LIN {X 0,Y 230.578,Z 317.111,A -85,B 0,C 180,E1 -20760.813,E2 -20760.813} C_VEL
LIN {X 0,Y 233.907,Z 325.789,A -85,B 0,C 180,E1 -20762.609,E2 -20762.609} C_VEL
LIN {X 0,Y 238.982,Z 335.486,A -85,B 0,C 180,E1 -20765.008,E2 -20765.008} C_VEL
LIN {X 0,Y 245.081,Z 344.302,A -85,B 0,C 180,E1 -20767.553,E2 -20767.553} C_VEL
LIN {X 0,Y 253.175,Z 353.284,A -85,B 0,C 180,E1 -20770.543,E2 -20770.543} C_VEL
LIN {X 0,Y 261.948,Z 361.164,A -85,B 0,C 180,E1 -20773.525,E2 -20773.525} C_VEL
LIN {X 0,Y 271.147,Z 368.091,A -85,B 0,C 180,E1 -20776.51,E2 -20776.51} C_VEL
LIN {X 0,Y 276.4,Z 371.69,A -85,B 0,C 180,E1 -20778.264,E2 -20778.264} C_VEL
LIN {X 0,Y 283.012,Z 376.04,A -85,B 0,C 180,E1 -20780.657,E2 -20780.657} C_VEL
LIN {X 0,Y 288.749,Z 379.536,A -85,B 0,C 180,E1 -20783.01,E2 -20783.01} C_VEL
LIN {X 0,Y 291.205,Z 381.266,A -85,B 0,C 180,E1 -20784.46,E2 -20784.46} C_VEL
LIN {X 0,Y 293.286,Z 382.591,A -85,B 0,C 180,E1 -20785.878,E2 -20785.878} C_VEL
LIN {X 0,Y 295.421,Z 383.606,A -85,B 0,C 180,E1 -20787.399,E2 -20787.399} C_VEL
LIN {X 0,Y 296.734,Z 384.085,A -85,B 0,C 180,E1 -20788.643,E2 -20788.643} C_VEL
LIN {X 0,Y 297.612,Z 384.263,A -85,B 0,C 180,E1 -20790,E2 -20790} C_VEL
LIN {X 0,Y 296.714,Z 384.086,A -85,B 0,C 180,E1 -20791.357,E2 -20791.357} C_VEL
LIN {X 0,Y 295.23,Z 383.531,A -85,B 0,C 180,E1 -20792.729,E2 -20792.729} C_VEL
LIN {X 0,Y 293.276,Z 382.591,A -85,B 0,C 180,E1 -20794.123,E2 -20794.123} C_VEL
LIN {X 0,Y 289.886,Z 380.295,A -85,B 0,C 180,E1 -20796.383,E2 -20796.383} C_VEL
LIN {X 0,Y 287.004,Z 378.499,A -85,B 0,C 180,E1 -20797.74,E2 -20797.74} C_VEL
LIN {X 0,Y 281.117,Z 374.761,A -85,B 0,C 180,E1 -20800.078,E2 -20800.078} C_VEL
LIN {X 0,Y 273.672,Z 369.778,A -85,B 0,C 180,E1 -20802.671,E2 -20802.671} C_VEL
LIN {X 0,Y 265.413,Z 363.851,A -85,B 0,C 180,E1 -20805.354,E2 -20805.354} C_VEL
LIN {X 0,Y 255.737,Z 355.726,A -85,B 0,C 180,E1 -20808.579,E2 -20808.579} C_VEL
LIN {X 0,Y 247.025,Z 346.636,A -85,B 0,C 180,E1 -20811.706,E2 -20811.706} C_VEL
LIN {X 0,Y 241.827,Z 339.902,A -85,B 0,C 180,E1 -20813.764,E2 -20813.764} C_VEL
LIN {X 0,Y 236.613,Z 331.326,A -85,B 0,C 180,E1 -20816.068,E2 -20816.068} C_VEL
LIN {X 0,Y 232.585,Z 322.649,A -85,B 0,C 180,E1 -20818.071,E2 -20818.071} C_VEL
LIN {X 0,Y 229.455,Z 313.908,A -85,B 0,C 180,E1 -20819.786,E2 -20819.786} C_VEL
LIN {X 0,Y 225.733,Z 303.804,A -85,B 0,C 180,E1 -20821.564,E2 -20821.564} C_VEL
LIN {X 0,Y 220.845,Z 293.133,A -85,B 0,C 180,E1 -20823.371,E2 -20823.371} C_VEL
LIN {X 0,Y 216.792,Z 285.655,A -85,B 0,C 180,E1 -20824.644,E2 -20824.644} C_VEL
LIN {X 0,Y 215.273,Z 282.957,A -85,B 0,C 180,E1 -20825.085,E2 -20825.085} C_VEL
LIN {X 0,Y 213.929,Z 280.441,A -85,B 0,C 180,E1 -20825.467,E2 -20825.467} C_VEL
LIN {X 0,Y 213.702,Z 279.367,A -85,B 0,C 180,E1 -20825.598,E2 -20825.598} C_VEL
LIN {X 0,Y 213.74,Z 279.361,A -85,B 0,C 180,E1 -20828.662,E2 -20828.662} C_VEL
LIN {X 0,Y 213.756,Z 279.358,A -85,B 0,C 180,E1 -20831.114,E2 -20831.114} C_VEL
LIN {X 0,Y 213.798,Z 279.354,A -85,B 0,C 180,E1 -20833.701,E2 -20833.701} C_VEL
LIN {X 0,Y 213.775,Z 279.356,A -85,B 0,C 180,E1 -20836.358,E2 -20836.358} C_VEL
LIN {X 0,Y 213.762,Z 279.358,A -85,B 0,C 180,E1 -20839.128,E2 -20839.128} C_VEL
LIN {X 0,Y 213.721,Z 279.363,A -85,B 0,C 180,E1 -20843.724,E2 -20843.724} C_VEL
LIN {X 0,Y 213.732,Z 279.361,A -85,B 0,C 180,E1 -20848.272,E2 -20848.272} C_VEL
LIN {X 0,Y 213.801,Z 279.352,A -85,B 0,C 180,E1 -20852.614,E2 -20852.614} C_VEL
LIN {X 0,Y 213.778,Z 279.355,A -85,B 0,C 180,E1 -20856.997,E2 -20856.997} C_VEL
LIN {X 0,Y 213.866,Z 279.345,A -85,B 0,C 180,E1 -20862.81,E2 -20862.81} C_VEL
LIN {X 0,Y 213.916,Z 279.336,A -85,B 0,C 180,E1 -20866.716,E2 -20866.716} C_VEL
LIN {X 0,Y 214.123,Z 279.307,A -85,B 0,C 180,E1 -20870.566,E2 -20870.566} C_VEL
LIN {X 0,Y 214.079,Z 279.318,A -85,B 0,C 180,E1 -20874.359,E2 -20874.359} C_VEL
LIN {X 0,Y 214.434,Z 279.246,A -85,B 0,C 180,E1 -20878.133,E2 -20878.133} C_VEL
LIN {X 0,Y 214.534,Z 279.246,A -85,B 0,C 180,E1 -20880.011,E2 -20880.011} C_VEL
LIN {X 0,Y 214.403,Z 279.274,A -85,B 0,C 180,E1 -20881.889,E2 -20881.889} C_VEL
LIN {X 0,Y 214.185,Z 279.305,A -85,B 0,C 180,E1 -20887.552,E2 -20887.552} C_VEL
LIN {X 0,Y 213.994,Z 279.33,A -85,B 0,C 180,E1 -20891.375,E2 -20891.375} C_VEL
LIN {X 0,Y 213.901,Z 279.342,A -85,B 0,C 180,E1 -20895.25,E2 -20895.25} C_VEL
LIN {X 0,Y 213.802,Z 279.353,A -85,B 0,C 180,E1 -20899.201,E2 -20899.201} C_VEL
LIN {X 0,Y 213.795,Z 279.355,A -85,B 0,C 180,E1 -20903.243,E2 -20903.243} C_VEL
LIN {X 0,Y 213.805,Z 279.532,A -85,B 0,C 180,E1 -20907.439,E2 -20907.439} C_VEL
LIN {X 0,Y 214.004,Z 281.177,A -85,B 0,C 180,E1 -20911.709,E2 -20911.709} C_VEL
LIN {X 0,Y 214.25,Z 283.111,A -85,B 0,C 180,E1 -20916.2,E2 -20916.2} C_VEL
LIN {X 0,Y 214.622,Z 285.39,A -85,B 0,C 180,E1 -20920.925,E2 -20920.925} C_VEL
LIN {X 0,Y 214.75,Z 286.989,A -85,B 0,C 180,E1 -20923.949,E2 -20923.949} C_VEL
LIN {X 0,Y 214.684,Z 288.477,A -85,B 0,C 180,E1 -20926.571,E2 -20926.571} C_VEL
LIN {X 0,Y 214.492,Z 289.965,A -85,B 0,C 180,E1 -20929.058,E2 -20929.058} C_VEL
LIN {X 0,Y 213.761,Z 292.894,A -85,B 0,C 180,E1 -20933.716,E2 -20933.716} C_VEL
LIN {X 0,Y 213.629,Z 293.565,A -85,B 0,C 180,E1 -20934.675,E2 -20934.675} C_VEL
LIN {X 0,Y 214.491,Z 296.709,A -85,B 0,C 180,E1 -20935.014,E2 -20935.014} C_VEL
LIN {X 0,Y 218.05,Z 307.158,A -85,B 0,C 180,E1 -20936.47,E2 -20936.47} C_VEL
LIN {X 0,Y 221.031,Z 319.519,A -85,B 0,C 180,E1 -20938.304,E2 -20938.304} C_VEL
LIN {X 0,Y 222.724,Z 329.353,A -85,B 0,C 180,E1 -20939.908,E2 -20939.908} C_VEL
LIN {X 0,Y 223.702,Z 338.852,A -85,B 0,C 180,E1 -20941.618,E2 -20941.618} C_VEL
LIN {X 0,Y 223.928,Z 348.013,A -85,B 0,C 180,E1 -20943.452,E2 -20943.452} C_VEL
LIN {X 0,Y 223.641,Z 352.493,A -85,B 0,C 180,E1 -20944.4,E2 -20944.4} C_VEL
LIN {X 0,Y 220.928,Z 362.07,A -85,B 0,C 180,E1 -20946.57,E2 -20946.57} C_VEL
LIN {X 0,Y 218.712,Z 369.736,A -85,B 0,C 180,E1 -20948.75,E2 -20948.75} C_VEL
LIN {X 0,Y 216.744,Z 376.438,A -85,B 0,C 180,E1 -20951.08,E2 -20951.08} C_VEL
LIN {X 0,Y 215.21,Z 381.639,A -85,B 0,C 180,E1 -20953.264,E2 -20953.264} C_VEL
LIN {X 0,Y 213.669,Z 384.495,A -85,B 0,C 180,E1 -20954.603,E2 -20954.603} C_VEL
LIN {X 0,Y 209.677,Z 388.477,A -85,B 0,C 180,E1 -20956.803,E2 -20956.803} C_VEL
LIN {X 0,Y 205.968,Z 391.837,A -85,B 0,C 180,E1 -20959.161,E2 -20959.161} C_VEL
LIN {X 0,Y 204.897,Z 393.47,A -85,B 0,C 180,E1 -20960.715,E2 -20960.715} C_VEL
LIN {X 0,Y 204.385,Z 396.131,A -85,B 0,C 180,E1 -20964.079,E2 -20964.079} C_VEL
LIN {X 0,Y 204.286,Z 397.242,A -85,B 0,C 180,E1 -20966.215,E2 -20966.215} C_VEL
LIN {X 0,Y 204.337,Z 397.788,A -85,B 0,C 180,E1 -20968.029,E2 -20968.029} C_VEL
LIN {X 0,Y 204.427,Z 397.946,A -85,B 0,C 180,E1 -20970,E2 -20970} C_VEL
LIN {X 0,Y 204.339,Z 397.788,A -85,B 0,C 180,E1 -20971.971,E2 -20971.971} C_VEL
LIN {X 0,Y 204.324,Z 397.195,A -85,B 0,C 180,E1 -20973.945,E2 -20973.945} C_VEL
LIN {X 0,Y 204.63,Z 394.739,A -85,B 0,C 180,E1 -20977.896,E2 -20977.896} C_VEL
LIN {X 0,Y 205.297,Z 391.785,A -85,B 0,C 180,E1 -20980.852,E2 -20980.852} C_VEL
LIN {X 0,Y 206.317,Z 387.79,A -85,B 0,C 180,E1 -20983.795,E2 -20983.795} C_VEL
LIN {X 0,Y 207.961,Z 382.661,A -85,B 0,C 180,E1 -20986.693,E2 -20986.693} C_VEL
LIN {X 0,Y 209.626,Z 377.398,A -85,B 0,C 180,E1 -20989.079,E2 -20989.079} C_VEL
LIN {X 0,Y 211.306,Z 372.46,A -85,B 0,C 180,E1 -20990.949,E2 -20990.949} C_VEL
LIN {X 0,Y 212.922,Z 366.757,A -85,B 0,C 180,E1 -20992.819,E2 -20992.819} C_VEL
LIN {X 0,Y 215.437,Z 358.203,A -85,B 0,C 180,E1 -20995.092,E2 -20995.092} C_VEL
LIN {X 0,Y 217.134,Z 352.295,A -85,B 0,C 180,E1 -20996.426,E2 -20996.426} C_VEL
LIN {X 0,Y 217.273,Z 342.791,A -85,B 0,C 180,E1 -20998.497,E2 -20998.497} C_VEL
LIN {X 0,Y 216.572,Z 333.544,A -85,B 0,C 180,E1 -21000.318,E2 -21000.318} C_VEL
LIN {X 0,Y 215.367,Z 324.393,A -85,B 0,C 180,E1 -21001.942,E2 -21001.942} C_VEL
LIN {X 0,Y 213.24,Z 314.25,A -85,B 0,C 180,E1 -21003.606,E2 -21003.606} C_VEL
LIN {X 0,Y 210.366,Z 304.243,A -85,B 0,C 180,E1 -21005.152,E2 -21005.152} C_VEL
LIN {X 0,Y 207.811,Z 296.964,A -85,B 0,C 180,E1 -21006.254,E2 -21006.254} C_VEL
LIN {X 0,Y 206.779,Z 293.718,A -85,B 0,C 180,E1 -21006.652,E2 -21006.652} C_VEL
LIN {X 0,Y 206.776,Z 293.334,A -85,B 0,C 180,E1 -21006.834,E2 -21006.834} C_VEL
LIN {X 0,Y 207.26,Z 291.24,A -85,B 0,C 180,E1 -21010.11,E2 -21010.11} C_VEL
LIN {X 0,Y 207.535,Z 289.738,A -85,B 0,C 180,E1 -21012.63,E2 -21012.63} C_VEL
LIN {X 0,Y 207.673,Z 288.273,A -85,B 0,C 180,E1 -21015.288,E2 -21015.288} C_VEL
LIN {X 0,Y 207.61,Z 286.781,A -85,B 0,C 180,E1 -21018.135,E2 -21018.135} C_VEL
LIN {X 0,Y 207.328,Z 284.754,A -85,B 0,C 180,E1 -21022.387,E2 -21022.387} C_VEL
LIN {X 0,Y 207.025,Z 282.704,A -85,B 0,C 180,E1 -21027.09,E2 -21027.09} C_VEL
LIN {X 0,Y 206.805,Z 280.99,A -85,B 0,C 180,E1 -21031.579,E2 -21031.579} C_VEL
LIN {X 0,Y 206.694,Z 280.24,A -85,B 0,C 180,E1 -21033.756,E2 -21033.756} C_VEL
LIN {X 0,Y 206.724,Z 280.238,A -85,B 0,C 180,E1 -21038.029,E2 -21038.029} C_VEL
LIN {X 0,Y 206.829,Z 280.223,A -85,B 0,C 180,E1 -21042.182,E2 -21042.182} C_VEL
LIN {X 0,Y 206.876,Z 280.216,A -85,B 0,C 180,E1 -21046.232,E2 -21046.232} C_VEL
LIN {X 0,Y 207.08,Z 280.189,A -85,B 0,C 180,E1 -21050.219,E2 -21050.219} C_VEL
LIN {X 0,Y 207.041,Z 280.194,A -85,B 0,C 180,E1 -21054.144,E2 -21054.144} C_VEL
LIN {X 0,Y 207.343,Z 280.153,A -85,B 0,C 180,E1 -21058.046,E2 -21058.046} C_VEL
LIN {X 0,Y 207.499,Z 280.12,A -85,B 0,C 180,E1 -21059.989,E2 -21059.989} C_VEL
LIN {X 0,Y 207.37,Z 280.124,A -85,B 0,C 180,E1 -21061.931,E2 -21061.931} C_VEL
LIN {X 0,Y 207.12,Z 280.183,A -85,B 0,C 180,E1 -21067.789,E2 -21067.789} C_VEL
LIN {X 0,Y 206.9,Z 280.212,A -85,B 0,C 180,E1 -21071.747,E2 -21071.747} C_VEL
LIN {X 0,Y 206.806,Z 280.221,A -85,B 0,C 180,E1 -21075.763,E2 -21075.763} C_VEL
LIN {X 0,Y 206.695,Z 280.23,A -85,B 0,C 180,E1 -21079.865,E2 -21079.865} C_VEL
LIN {X 0,Y 206.717,Z 280.232,A -85,B 0,C 180,E1 -21084.064,E2 -21084.064} C_VEL
LIN {X 0,Y 206.701,Z 280.237,A -85,B 0,C 180,E1 -21088.41,E2 -21088.41} C_VEL
LIN {X 0,Y 206.672,Z 280.239,A -85,B 0,C 180,E1 -21092.947,E2 -21092.947} C_VEL
LIN {X 0,Y 206.692,Z 280.239,A -85,B 0,C 180,E1 -21097.72,E2 -21097.72} C_VEL
LIN {X 0,Y 206.69,Z 280.239,A -85,B 0,C 180,E1 -21101.579,E2 -21101.579} C_VEL
LIN {X 0,Y 206.708,Z 280.235,A -85,B 0,C 180,E1 -21105.541,E2 -21105.541} C_VEL
LIN {X 0,Y 206.685,Z 280.238,A -85,B 0,C 180,E1 -21109.756,E2 -21109.756} C_VEL
LIN {X 0,Y 206.681,Z 280.24,A -85,B 0,C 180,E1 -21113.047,E2 -21113.047} C_VEL
LIN {X 0,Y 207.723,Z 283.16,A -85,B 0,C 180,E1 -21113.46,E2 -21113.46} C_VEL
LIN {X 0,Y 209.099,Z 285.173,A -85,B 0,C 180,E1 -21113.852,E2 -21113.852} C_VEL
LIN {X 0,Y 215.11,Z 296.436,A -85,B 0,C 180,E1 -21115.873,E2 -21115.873} C_VEL
LIN {X 0,Y 220.512,Z 308.717,A -85,B 0,C 180,E1 -21118.145,E2 -21118.145} C_VEL
LIN {X 0,Y 224.337,Z 319.993,A -85,B 0,C 180,E1 -21120.337,E2 -21120.337} C_VEL
LIN {X 0,Y 227.363,Z 328.293,A -85,B 0,C 180,E1 -21122.168,E2 -21122.168} C_VEL
LIN {X 0,Y 230.978,Z 335.793,A -85,B 0,C 180,E1 -21124.091,E2 -21124.091} C_VEL
LIN {X 0,Y 236.873,Z 345.062,A -85,B 0,C 180,E1 -21126.858,E2 -21126.858} C_VEL
LIN {X 0,Y 242.506,Z 351.873,A -85,B 0,C 180,E1 -21129.176,E2 -21129.176} C_VEL
LIN {X 0,Y 250.815,Z 359.906,A -85,B 0,C 180,E1 -21132.266,E2 -21132.266} C_VEL
LIN {X 0,Y 258.387,Z 365.909,A -85,B 0,C 180,E1 -21134.873,E2 -21134.873} C_VEL
LIN {X 0,Y 266.288,Z 371.277,A -85,B 0,C 180,E1 -21137.503,E2 -21137.503} C_VEL
LIN {X 0,Y 272.247,Z 375.005,A -85,B 0,C 180,E1 -21139.59,E2 -21139.59} C_VEL
LIN {X 0,Y 277.139,Z 377.882,A -85,B 0,C 180,E1 -21141.416,E2 -21141.416} C_VEL
LIN {X 0,Y 280.561,Z 379.762,A -85,B 0,C 180,E1 -21142.805,E2 -21142.805} C_VEL
LIN {X 0,Y 283.586,Z 381.477,A -85,B 0,C 180,E1 -21144.311,E2 -21144.311} C_VEL
LIN {X 0,Y 285.742,Z 382.797,A -85,B 0,C 180,E1 -21145.769,E2 -21145.769} C_VEL
LIN {X 0,Y 288.344,Z 383.933,A -85,B 0,C 180,E1 -21147.589,E2 -21147.589} C_VEL
LIN {X 0,Y 289.446,Z 384.284,A -85,B 0,C 180,E1 -21148.609,E2 -21148.609} C_VEL
LIN {X 0,Y 290.46,Z 384.455,A -85,B 0,C 180,E1 -21150,E2 -21150} C_VEL
LIN {X 0,Y 289.429,Z 384.285,A -85,B 0,C 180,E1 -21151.391,E2 -21151.391} C_VEL
LIN {X 0,Y 287.789,Z 383.737,A -85,B 0,C 180,E1 -21152.799,E2 -21152.799} C_VEL
LIN {X 0,Y 285.735,Z 382.797,A -85,B 0,C 180,E1 -21154.232,E2 -21154.232} C_VEL
LIN {X 0,Y 282.715,Z 380.938,A -85,B 0,C 180,E1 -21156.199,E2 -21156.199} C_VEL
LIN {X 0,Y 280.563,Z 379.762,A -85,B 0,C 180,E1 -21157.195,E2 -21157.195} C_VEL
LIN {X 0,Y 274.632,Z 376.375,A -85,B 0,C 180,E1 -21159.575,E2 -21159.575} C_VEL
LIN {X 0,Y 267.397,Z 371.944,A -85,B 0,C 180,E1 -21162.138,E2 -21162.138} C_VEL
LIN {X 0,Y 258.395,Z 365.888,A -85,B 0,C 180,E1 -21165.134,E2 -21165.134} C_VEL
LIN {X 0,Y 250.083,Z 359.226,A -85,B 0,C 180,E1 -21168.006,E2 -21168.006} C_VEL
LIN {X 0,Y 242.532,Z 351.852,A -85,B 0,C 180,E1 -21170.828,E2 -21170.828} C_VEL
LIN {X 0,Y 235.805,Z 343.591,A -85,B 0,C 180,E1 -21173.617,E2 -21173.617} C_VEL
LIN {X 0,Y 230.422,Z 334.739,A -85,B 0,C 180,E1 -21176.19,E2 -21176.19} C_VEL
LIN {X 0,Y 226.467,Z 325.993,A -85,B 0,C 180,E1 -21178.376,E2 -21178.376} C_VEL
LIN {X 0,Y 222.659,Z 314.815,A -85,B 0,C 180,E1 -21180.697,E2 -21180.697} C_VEL
LIN {X 0,Y 219.223,Z 305.511,A -85,B 0,C 180,E1 -21182.452,E2 -21182.452} C_VEL
LIN {X 0,Y 213.984,Z 294.191,A -85,B 0,C 180,E1 -21184.52,E2 -21184.52} C_VEL
LIN {X 0,Y 208.49,Z 284.179,A -85,B 0,C 180,E1 -21186.346,E2 -21186.346} C_VEL
LIN {X 0,Y 207.06,Z 281.823,A -85,B 0,C 180,E1 -21186.774,E2 -21186.774} C_VEL
LIN {X 0,Y 206.668,Z 280.242,A -85,B 0,C 180,E1 -21186.948,E2 -21186.948} C_VEL
LIN {X 0,Y 206.685,Z 280.24,A -85,B 0,C 180,E1 -21191.597,E2 -21191.597} C_VEL
LIN {X 0,Y 206.709,Z 280.236,A -85,B 0,C 180,E1 -21195.559,E2 -21195.559} C_VEL
LIN {X 0,Y 206.692,Z 280.238,A -85,B 0,C 180,E1 -21199.774,E2 -21199.774} C_VEL
LIN {X 0,Y 206.692,Z 280.239,A -85,B 0,C 180,E1 -21202.28,E2 -21202.28} C_VEL
LIN {X 0,Y 206.672,Z 280.239,A -85,B 0,C 180,E1 -21207.053,E2 -21207.053} C_VEL
LIN {X 0,Y 206.727,Z 280.234,A -85,B 0,C 180,E1 -21212.115,E2 -21212.115} C_VEL
LIN {X 0,Y 206.719,Z 280.233,A -85,B 0,C 180,E1 -21216.624,E2 -21216.624} C_VEL
LIN {X 0,Y 206.804,Z 280.224,A -85,B 0,C 180,E1 -21222.203,E2 -21222.203} C_VEL
LIN {X 0,Y 206.856,Z 280.214,A -85,B 0,C 180,E1 -21226.254,E2 -21226.254} C_VEL
LIN {X 0,Y 207.067,Z 280.185,A -85,B 0,C 180,E1 -21230.242,E2 -21230.242} C_VEL
LIN {X 0,Y 207.04,Z 280.194,A -85,B 0,C 180,E1 -21234.167,E2 -21234.167} C_VEL
LIN {X 0,Y 207.37,Z 280.124,A -85,B 0,C 180,E1 -21238.069,E2 -21238.069} C_VEL
LIN {X 0,Y 207.499,Z 280.12,A -85,B 0,C 180,E1 -21240.011,E2 -21240.011} C_VEL
LIN {X 0,Y 207.044,Z 280.194,A -85,B 0,C 180,E1 -21243.904,E2 -21243.904} C_VEL
LIN {X 0,Y 207.129,Z 280.184,A -85,B 0,C 180,E1 -21247.811,E2 -21247.811} C_VEL
LIN {X 0,Y 206.917,Z 280.212,A -85,B 0,C 180,E1 -21251.77,E2 -21251.77} C_VEL
LIN {X 0,Y 206.829,Z 280.224,A -85,B 0,C 180,E1 -21255.784,E2 -21255.784} C_VEL
LIN {X 0,Y 206.723,Z 280.235,A -85,B 0,C 180,E1 -21259.886,E2 -21259.886} C_VEL
LIN {X 0,Y 206.732,Z 280.236,A -85,B 0,C 180,E1 -21264.087,E2 -21264.087} C_VEL
LIN {X 0,Y 206.702,Z 280.239,A -85,B 0,C 180,E1 -21266.243,E2 -21266.243} C_VEL
LIN {X 0,Y 206.925,Z 281.813,A -85,B 0,C 180,E1 -21270.639,E2 -21270.639} C_VEL
LIN {X 0,Y 207.186,Z 283.821,A -85,B 0,C 180,E1 -21275.502,E2 -21275.502} C_VEL
LIN {X 0,Y 207.501,Z 285.905,A -85,B 0,C 180,E1 -21280.067,E2 -21280.067} C_VEL
LIN {X 0,Y 207.628,Z 287.177,A -85,B 0,C 180,E1 -21282.62,E2 -21282.62} C_VEL
LIN {X 0,Y 207.662,Z 288.619,A -85,B 0,C 180,E1 -21285.305,E2 -21285.305} C_VEL
LIN {X 0,Y 207.472,Z 290.265,A -85,B 0,C 180,E1 -21288.193,E2 -21288.193} C_VEL
LIN {X 0,Y 206.907,Z 292.7,A -85,B 0,C 180,E1 -21292.31,E2 -21292.31} C_VEL
LIN {X 0,Y 206.759,Z 293.35,A -85,B 0,C 180,E1 -21293.28,E2 -21293.28} C_VEL
LIN {X 0,Y 207.689,Z 296.641,A -85,B 0,C 180,E1 -21293.7,E2 -21293.7} C_VEL
LIN {X 0,Y 211.588,Z 307.857,A -85,B 0,C 180,E1 -21295.393,E2 -21295.393} C_VEL
LIN {X 0,Y 214.327,Z 319.137,A -85,B 0,C 180,E1 -21297.167,E2 -21297.167} C_VEL
LIN {X 0,Y 216.088,Z 329.141,A -85,B 0,C 180,E1 -21298.883,E2 -21298.883} C_VEL
LIN {X 0,Y 216.987,Z 338.103,A -85,B 0,C 180,E1 -21300.55,E2 -21300.55} C_VEL
LIN {X 0,Y 217.319,Z 346.098,A -85,B 0,C 180,E1 -21302.187,E2 -21302.187} C_VEL
LIN {X 0,Y 216.95,Z 353.387,A -85,B 0,C 180,E1 -21303.809,E2 -21303.809} C_VEL
LIN {X 0,Y 214.401,Z 361.875,A -85,B 0,C 180,E1 -21305.812,E2 -21305.812} C_VEL
LIN {X 0,Y 211.872,Z 370.183,A -85,B 0,C 180,E1 -21308.267,E2 -21308.267} C_VEL
LIN {X 0,Y 210.028,Z 376.243,A -85,B 0,C 180,E1 -21310.451,E2 -21310.451} C_VEL
LIN {X 0,Y 208.266,Z 381.795,A -85,B 0,C 180,E1 -21312.875,E2 -21312.875} C_VEL
LIN {X 0,Y 206.822,Z 386.237,A -85,B 0,C 180,E1 -21315.235,E2 -21315.235} C_VEL
LIN {X 0,Y 205.592,Z 390.565,A -85,B 0,C 180,E1 -21318.165,E2 -21318.165} C_VEL
LIN {X 0,Y 204.897,Z 393.47,A -85,B 0,C 180,E1 -21320.715,E2 -21320.715} C_VEL
LIN {X 0,Y 203.924,Z 394.935,A -85,B 0,C 180,E1 -21322.305,E2 -21322.305} C_VEL
LIN {X 0,Y 200.778,Z 396.597,A -85,B 0,C 180,E1 -21324.928,E2 -21324.928} C_VEL
LIN {X 0,Y 198.306,Z 397.369,A -85,B 0,C 180,E1 -21327.097,E2 -21327.097} C_VEL
LIN {X 0,Y 197.324,Z 397.75,A -85,B 0,C 180,E1 -21328.795,E2 -21328.795} C_VEL
LIN {X 0,Y 197.277,Z 397.703,A -85,B 0,C 180,E1 -21329.37,E2 -21329.37} C_VEL
LIN {X 0,Y 197.247,Z 397.593,A -85,B 0,C 180,E1 -21332.042,E2 -21332.042} C_VEL
LIN {X 0,Y 197.234,Z 397,A -85,B 0,C 180,E1 -21334.087,E2 -21334.087} C_VEL
LIN {X 0,Y 197.567,Z 394.543,A -85,B 0,C 180,E1 -21338.18,E2 -21338.18} C_VEL
LIN {X 0,Y 198.287,Z 391.589,A -85,B 0,C 180,E1 -21341.241,E2 -21341.241} C_VEL
LIN {X 0,Y 199.392,Z 387.595,A -85,B 0,C 180,E1 -21344.284,E2 -21344.284} C_VEL
LIN {X 0,Y 201.148,Z 382.465,A -85,B 0,C 180,E1 -21347.276,E2 -21347.276} C_VEL
LIN {X 0,Y 202.913,Z 377.203,A -85,B 0,C 180,E1 -21349.736,E2 -21349.736} C_VEL
LIN {X 0,Y 204.639,Z 372.273,A -85,B 0,C 180,E1 -21351.662,E2 -21351.662} C_VEL
LIN {X 0,Y 206.362,Z 366.561,A -85,B 0,C 180,E1 -21353.587,E2 -21353.587} C_VEL
LIN {X 0,Y 209.019,Z 358.008,A -85,B 0,C 180,E1 -21355.919,E2 -21355.919} C_VEL
LIN {X 0,Y 210.472,Z 353.188,A -85,B 0,C 180,E1 -21357.062,E2 -21357.062} C_VEL
LIN {X 0,Y 210.664,Z 342.583,A -85,B 0,C 180,E1 -21359.478,E2 -21359.478} C_VEL
LIN {X 0,Y 209.919,Z 332.761,A -85,B 0,C 180,E1 -21361.483,E2 -21361.483} C_VEL
LIN {X 0,Y 208.634,Z 323.932,A -85,B 0,C 180,E1 -21363.136,E2 -21363.136} C_VEL
LIN {X 0,Y 206.635,Z 314.374,A -85,B 0,C 180,E1 -21364.793,E2 -21364.793} C_VEL
LIN {X 0,Y 203.646,Z 304.117,A -85,B 0,C 180,E1 -21366.486,E2 -21366.486} C_VEL
LIN {X 0,Y 200.911,Z 296.641,A -85,B 0,C 180,E1 -21367.717,E2 -21367.717} C_VEL
LIN {X 0,Y 199.958,Z 293.545,A -85,B 0,C 180,E1 -21368.117,E2 -21368.117} C_VEL
LIN {X 0,Y 199.948,Z 293.096,A -85,B 0,C 180,E1 -21368.36,E2 -21368.36} C_VEL
LIN {X 0,Y 200.486,Z 290.582,A -85,B 0,C 180,E1 -21372.582,E2 -21372.582} C_VEL
LIN {X 0,Y 200.617,Z 289.021,A -85,B 0,C 180,E1 -21375.509,E2 -21375.509} C_VEL
LIN {X 0,Y 200.577,Z 287.643,A -85,B 0,C 180,E1 -21378.249,E2 -21378.249} C_VEL
LIN {X 0,Y 200.393,Z 286.44,A -85,B 0,C 180,E1 -21380.843,E2 -21380.843} C_VEL
LIN {X 0,Y 200.071,Z 284.295,A -85,B 0,C 180,E1 -21385.791,E2 -21385.791} C_VEL
LIN {X 0,Y 199.814,Z 282.461,A -85,B 0,C 180,E1 -21390.489,E2 -21390.489} C_VEL
LIN {X 0,Y 199.646,Z 281.119,A -85,B 0,C 180,E1 -21395.001,E2 -21395.001} C_VEL
LIN {X 0,Y 199.655,Z 281.119,A -85,B 0,C 180,E1 -21399.379,E2 -21399.379} C_VEL
LIN {X 0,Y 199.767,Z 281.103,A -85,B 0,C 180,E1 -21403.642,E2 -21403.642} C_VEL
LIN {X 0,Y 199.867,Z 281.09,A -85,B 0,C 180,E1 -21407.809,E2 -21407.809} C_VEL
LIN {X 0,Y 200.077,Z 281.063,A -85,B 0,C 180,E1 -21411.912,E2 -21411.912} C_VEL
LIN {X 0,Y 200.285,Z 281.033,A -85,B 0,C 180,E1 -21417.977,E2 -21417.977} C_VEL
LIN {X 0,Y 200.463,Z 280.995,A -85,B 0,C 180,E1 -21419.988,E2 -21419.988} C_VEL
LIN {X 0,Y 200.008,Z 281.056,A -85,B 0,C 180,E1 -21424.018,E2 -21424.018} C_VEL
LIN {X 0,Y 200.067,Z 281.062,A -85,B 0,C 180,E1 -21428.065,E2 -21428.065} C_VEL
LIN {X 0,Y 199.849,Z 281.09,A -85,B 0,C 180,E1 -21432.168,E2 -21432.168} C_VEL
LIN {X 0,Y 199.744,Z 281.102,A -85,B 0,C 180,E1 -21436.335,E2 -21436.335} C_VEL
LIN {X 0,Y 199.627,Z 281.112,A -85,B 0,C 180,E1 -21440.599,E2 -21440.599} C_VEL
LIN {X 0,Y 199.637,Z 281.11,A -85,B 0,C 180,E1 -21444.974,E2 -21444.974} C_VEL
LIN {X 0,Y 199.63,Z 281.118,A -85,B 0,C 180,E1 -21449.514,E2 -21449.514} C_VEL
LIN {X 0,Y 199.622,Z 281.121,A -85,B 0,C 180,E1 -21452.335,E2 -21452.335} C_VEL
LIN {X 0,Y 199.621,Z 281.12,A -85,B 0,C 180,E1 -21456.746,E2 -21456.746} C_VEL
LIN {X 0,Y 199.645,Z 281.116,A -85,B 0,C 180,E1 -21459.301,E2 -21459.301} C_VEL
LIN {X 0,Y 199.628,Z 281.118,A -85,B 0,C 180,E1 -21462.328,E2 -21462.328} C_VEL
LIN {X 0,Y 199.656,Z 281.113,A -85,B 0,C 180,E1 -21465.252,E2 -21465.252} C_VEL
LIN {X 0,Y 199.628,Z 281.119,A -85,B 0,C 180,E1 -21468.019,E2 -21468.019} C_VEL
LIN {X 0,Y 199.666,Z 281.115,A -85,B 0,C 180,E1 -21471.546,E2 -21471.546} C_VEL
LIN {X 0,Y 200.835,Z 284.251,A -85,B 0,C 180,E1 -21472.041,E2 -21472.041} C_VEL
LIN {X 0,Y 202.221,Z 286.242,A -85,B 0,C 180,E1 -21472.463,E2 -21472.463} C_VEL
LIN {X 0,Y 208.635,Z 298.108,A -85,B 0,C 180,E1 -21474.801,E2 -21474.801} C_VEL
LIN {X 0,Y 213.942,Z 310.248,A -85,B 0,C 180,E1 -21477.229,E2 -21477.229} C_VEL
LIN {X 0,Y 217.028,Z 319.306,A -85,B 0,C 180,E1 -21479.08,E2 -21479.08} C_VEL
LIN {X 0,Y 219.926,Z 328.382,A -85,B 0,C 180,E1 -21481.114,E2 -21481.114} C_VEL
LIN {X 0,Y 223.951,Z 337.692,A -85,B 0,C 180,E1 -21483.592,E2 -21483.592} C_VEL
LIN {X 0,Y 228.946,Z 346.049,A -85,B 0,C 180,E1 -21486.2,E2 -21486.2} C_VEL
LIN {X 0,Y 234.062,Z 352.592,A -85,B 0,C 180,E1 -21488.525,E2 -21488.525} C_VEL
LIN {X 0,Y 240.827,Z 359.487,A -85,B 0,C 180,E1 -21491.276,E2 -21491.276} C_VEL
LIN {X 0,Y 248.414,Z 365.749,A -85,B 0,C 180,E1 -21494.088,E2 -21494.088} C_VEL
LIN {X 0,Y 255.837,Z 370.793,A -85,B 0,C 180,E1 -21496.652,E2 -21496.652} C_VEL
LIN {X 0,Y 264.331,Z 375.836,A -85,B 0,C 180,E1 -21499.588,E2 -21499.588} C_VEL
LIN {X 0,Y 269.876,Z 378.779,A -85,B 0,C 180,E1 -21501.637,E2 -21501.637} C_VEL
LIN {X 0,Y 275.776,Z 381.693,A -85,B 0,C 180,E1 -21504.149,E2 -21504.149} C_VEL
LIN {X 0,Y 278.185,Z 383.003,A -85,B 0,C 180,E1 -21505.653,E2 -21505.653} C_VEL
LIN {X 0,Y 281.27,Z 384.229,A -85,B 0,C 180,E1 -21507.792,E2 -21507.792} C_VEL
LIN {X 0,Y 282.154,Z 384.483,A -85,B 0,C 180,E1 -21508.573,E2 -21508.573} C_VEL
LIN {X 0,Y 283.294,Z 384.648,A -85,B 0,C 180,E1 -21510,E2 -21510} C_VEL
LIN {X 0,Y 282.141,Z 384.484,A -85,B 0,C 180,E1 -21511.427,E2 -21511.427} C_VEL
LIN {X 0,Y 280.287,Z 383.944,A -85,B 0,C 180,E1 -21512.874,E2 -21512.874} C_VEL
LIN {X 0,Y 278.182,Z 383.003,A -85,B 0,C 180,E1 -21514.347,E2 -21514.347} C_VEL
LIN {X 0,Y 275.531,Z 381.573,A -85,B 0,C 180,E1 -21515.975,E2 -21515.975} C_VEL
LIN {X 0,Y 269.881,Z 378.769,A -85,B 0,C 180,E1 -21518.369,E2 -21518.369} C_VEL
LIN {X 0,Y 264.336,Z 375.823,A -85,B 0,C 180,E1 -21520.418,E2 -21520.418} C_VEL
LIN {X 0,Y 258.13,Z 372.206,A -85,B 0,C 180,E1 -21522.58,E2 -21522.58} C_VEL
LIN {X 0,Y 250.446,Z 367.193,A -85,B 0,C 180,E1 -21525.215,E2 -21525.215} C_VEL
LIN {X 0,Y 242.119,Z 360.649,A -85,B 0,C 180,E1 -21528.232,E2 -21528.232} C_VEL
LIN {X 0,Y 235.123,Z 353.797,A -85,B 0,C 180,E1 -21531.019,E2 -21531.019} C_VEL
LIN {X 0,Y 229.702,Z 347.135,A -85,B 0,C 180,E1 -21533.437,E2 -21533.437} C_VEL
LIN {X 0,Y 224.788,Z 339.218,A -85,B 0,C 180,E1 -21535.957,E2 -21535.957} C_VEL
LIN {X 0,Y 221.142,Z 331.552,A -85,B 0,C 180,E1 -21538.091,E2 -21538.091} C_VEL
LIN {X 0,Y 218.2,Z 323.262,A -85,B 0,C 180,E1 -21540.075,E2 -21540.075} C_VEL
LIN {X 0,Y 214.953,Z 312.965,A -85,B 0,C 180,E1 -21542.216,E2 -21542.216} C_VEL
LIN {X 0,Y 211.054,Z 303.415,A -85,B 0,C 180,E1 -21544.14,E2 -21544.14} C_VEL
LIN {X 0,Y 206.452,Z 293.98,A -85,B 0,C 180,E1 -21546.009,E2 -21546.009} C_VEL
LIN {X 0,Y 201.986,Z 285.723,A -85,B 0,C 180,E1 -21547.63,E2 -21547.63} C_VEL
LIN {X 0,Y 200.14,Z 282.936,A -85,B 0,C 180,E1 -21548.221,E2 -21548.221} C_VEL
LIN {X 0,Y 199.666,Z 281.115,A -85,B 0,C 180,E1 -21548.467,E2 -21548.467} C_VEL
LIN {X 0,Y 199.624,Z 281.118,A -85,B 0,C 180,E1 -21552.347,E2 -21552.347} C_VEL
LIN {X 0,Y 199.657,Z 281.113,A -85,B 0,C 180,E1 -21555.271,E2 -21555.271} C_VEL
LIN {X 0,Y 199.632,Z 281.119,A -85,B 0,C 180,E1 -21558.038,E2 -21558.038} C_VEL
LIN {X 0,Y 199.647,Z 281.116,A -85,B 0,C 180,E1 -21560.753,E2 -21560.753} C_VEL
LIN {X 0,Y 199.601,Z 281.122,A -85,B 0,C 180,E1 -21565.728,E2 -21565.728} C_VEL
LIN {X 0,Y 199.66,Z 281.114,A -85,B 0,C 180,E1 -21568.146,E2 -21568.146} C_VEL
LIN {X 0,Y 199.653,Z 281.115,A -85,B 0,C 180,E1 -21572.782,E2 -21572.782} C_VEL
LIN {X 0,Y 199.658,Z 281.115,A -85,B 0,C 180,E1 -21577.234,E2 -21577.234} C_VEL
LIN {X 0,Y 199.727,Z 281.106,A -85,B 0,C 180,E1 -21581.815,E2 -21581.815} C_VEL
LIN {X 0,Y 199.794,Z 281.092,A -85,B 0,C 180,E1 -21585.758,E2 -21585.758} C_VEL
LIN {X 0,Y 200.011,Z 281.064,A -85,B 0,C 180,E1 -21589.894,E2 -21589.894} C_VEL
LIN {X 0,Y 200.003,Z 281.07,A -85,B 0,C 180,E1 -21593.961,E2 -21593.961} C_VEL
LIN {X 0,Y 200.31,Z 281.002,A -85,B 0,C 180,E1 -21598.001,E2 -21598.001} C_VEL
LIN {X 0,Y 200.463,Z 280.995,A -85,B 0,C 180,E1 -21600.012,E2 -21600.012} C_VEL
LIN {X 0,Y 199.991,Z 281.073,A -85,B 0,C 180,E1 -21604.042,E2 -21604.042} C_VEL
LIN {X 0,Y 200.077,Z 281.064,A -85,B 0,C 180,E1 -21608.088,E2 -21608.088} C_VEL
LIN {X 0,Y 199.867,Z 281.092,A -85,B 0,C 180,E1 -21612.191,E2 -21612.191} C_VEL
LIN {X 0,Y 199.767,Z 281.103,A -85,B 0,C 180,E1 -21616.358,E2 -21616.358} C_VEL
LIN {X 0,Y 199.655,Z 281.116,A -85,B 0,C 180,E1 -21620.621,E2 -21620.621} C_VEL
LIN {X 0,Y 199.648,Z 281.118,A -85,B 0,C 180,E1 -21624.999,E2 -21624.999} C_VEL
LIN {X 0,Y 199.814,Z 282.492,A -85,B 0,C 180,E1 -21629.511,E2 -21629.511} C_VEL
LIN {X 0,Y 200.071,Z 284.314,A -85,B 0,C 180,E1 -21634.209,E2 -21634.209} C_VEL
LIN {X 0,Y 200.422,Z 286.603,A -85,B 0,C 180,E1 -21639.517,E2 -21639.517} C_VEL
LIN {X 0,Y 200.582,Z 288.079,A -85,B 0,C 180,E1 -21642.627,E2 -21642.627} C_VEL
LIN {X 0,Y 200.6,Z 289.581,A -85,B 0,C 180,E1 -21645.518,E2 -21645.518} C_VEL
LIN {X 0,Y 200.396,Z 291.061,A -85,B 0,C 180,E1 -21648.216,E2 -21648.216} C_VEL
LIN {X 0,Y 199.929,Z 293.178,A -85,B 0,C 180,E1 -21651.842,E2 -21651.842} C_VEL
LIN {X 0,Y 200.795,Z 296.373,A -85,B 0,C 180,E1 -21652.239,E2 -21652.239} C_VEL
LIN {X 0,Y 201.73,Z 298.622,A -85,B 0,C 180,E1 -21652.627,E2 -21652.627} C_VEL
LIN {X 0,Y 205.439,Z 309.724,A -85,B 0,C 180,E1 -21654.44,E2 -21654.44} C_VEL
LIN {X 0,Y 207.892,Z 319.912,A -85,B 0,C 180,E1 -21656.157,E2 -21656.157} C_VEL
LIN {X 0,Y 209.597,Z 330.127,A -85,B 0,C 180,E1 -21658.012,E2 -21658.012} C_VEL
LIN {X 0,Y 210.444,Z 338.771,A -85,B 0,C 180,E1 -21659.718,E2 -21659.718} C_VEL
LIN {X 0,Y 210.708,Z 346.406,A -85,B 0,C 180,E1 -21661.357,E2 -21661.357} C_VEL
LIN {X 0,Y 210.502,Z 353.189,A -85,B 0,C 180,E1 -21662.942,E2 -21662.942} C_VEL
LIN {X 0,Y 207.91,Z 361.679,A -85,B 0,C 180,E1 -21665.006,E2 -21665.006} C_VEL
LIN {X 0,Y 205.391,Z 369.648,A -85,B 0,C 180,E1 -21667.414,E2 -21667.414} C_VEL
LIN {X 0,Y 203.343,Z 376.048,A -85,B 0,C 180,E1 -21669.781,E2 -21669.781} C_VEL
LIN {X 0,Y 201.858,Z 380.551,A -85,B 0,C 180,E1 -21671.739,E2 -21671.739} C_VEL
LIN {X 0,Y 199.923,Z 386.041,A -85,B 0,C 180,E1 -21674.714,E2 -21674.714} C_VEL
LIN {X 0,Y 198.616,Z 390.37,A -85,B 0,C 180,E1 -21677.743,E2 -21677.743} C_VEL
LIN {X 0,Y 197.82,Z 393.457,A -85,B 0,C 180,E1 -21680.588,E2 -21680.588} C_VEL
LIN {X 0,Y 197.314,Z 395.936,A -85,B 0,C 180,E1 -21683.866,E2 -21683.866} C_VEL
LIN {X 0,Y 197.205,Z 397.136,A -85,B 0,C 180,E1 -21686.384,E2 -21686.384} C_VEL
LIN {X 0,Y 197.277,Z 397.703,A -85,B 0,C 180,E1 -21689.37,E2 -21689.37} C_VEL
LIN {X 0,Y 196.659,Z 397.739,A -85,B 0,C 180,E1 -21691.071,E2 -21691.071} C_VEL
LIN {X 0,Y 195.057,Z 397.404,A -85,B 0,C 180,E1 -21692.741,E2 -21692.741} C_VEL
LIN {X 0,Y 191.361,Z 395.897,A -85,B 0,C 180,E1 -21696.103,E2 -21696.103} C_VEL
LIN {X 0,Y 190.496,Z 394.873,A -85,B 0,C 180,E1 -21697.851,E2 -21697.851} C_VEL
LIN {X 0,Y 190.516,Z 394.378,A -85,B 0,C 180,E1 -21698.44,E2 -21698.44} C_VEL
LIN {X 0,Y 191.3,Z 391.393,A -85,B 0,C 180,E1 -21701.657,E2 -21701.657} C_VEL
LIN {X 0,Y 192.482,Z 387.399,A -85,B 0,C 180,E1 -21704.808,E2 -21704.808} C_VEL
LIN {X 0,Y 194.358,Z 382.27,A -85,B 0,C 180,E1 -21707.9,E2 -21707.9} C_VEL
LIN {X 0,Y 196.236,Z 377.008,A -85,B 0,C 180,E1 -21710.437,E2 -21710.437} C_VEL
LIN {X 0,Y 198.039,Z 371.988,A -85,B 0,C 180,E1 -21712.458,E2 -21712.458} C_VEL
LIN {X 0,Y 199.84,Z 366.364,A -85,B 0,C 180,E1 -21714.407,E2 -21714.407} C_VEL
LIN {X 0,Y 202.654,Z 357.814,A -85,B 0,C 180,E1 -21716.797,E2 -21716.797} C_VEL
LIN {X 0,Y 203.899,Z 352.985,A -85,B 0,C 180,E1 -21718.009,E2 -21718.009} C_VEL
LIN {X 0,Y 204.152,Z 343.724,A -85,B 0,C 180,E1 -21720.234,E2 -21720.234} C_VEL
LIN {X 0,Y 203.436,Z 333.6,A -85,B 0,C 180,E1 -21722.421,E2 -21722.421} C_VEL
LIN {X 0,Y 201.99,Z 323.473,A -85,B 0,C 180,E1 -21724.411,E2 -21724.411} C_VEL
LIN {X 0,Y 200.071,Z 314.315,A -85,B 0,C 180,E1 -21726.09,E2 -21726.09} C_VEL
LIN {X 0,Y 196.857,Z 303.784,A -85,B 0,C 180,E1 -21727.971,E2 -21727.971} C_VEL
LIN {X 0,Y 194.37,Z 296.909,A -85,B 0,C 180,E1 -21729.184,E2 -21729.184} C_VEL
LIN {X 0,Y 193.196,Z 293.879,A -85,B 0,C 180,E1 -21729.672,E2 -21729.672} C_VEL
LIN {X 0,Y 193.078,Z 292.979,A -85,B 0,C 180,E1 -21729.807,E2 -21729.807} C_VEL
LIN {X 0,Y 193.467,Z 290.837,A -85,B 0,C 180,E1 -21733.645,E2 -21733.645} C_VEL
LIN {X 0,Y 193.537,Z 289.364,A -85,B 0,C 180,E1 -21736.573,E2 -21736.573} C_VEL
LIN {X 0,Y 193.418,Z 287.87,A -85,B 0,C 180,E1 -21739.732,E2 -21739.732} C_VEL
LIN {X 0,Y 193.116,Z 285.889,A -85,B 0,C 180,E1 -21744.376,E2 -21744.376} C_VEL
LIN {X 0,Y 192.998,Z 284.901,A -85,B 0,C 180,E1 -21746.879,E2 -21746.879} C_VEL
LIN {X 0,Y 192.766,Z 283.143,A -85,B 0,C 180,E1 -21751.696,E2 -21751.696} C_VEL
LIN {X 0,Y 192.637,Z 281.993,A -85,B 0,C 180,E1 -21755.791,E2 -21755.791} C_VEL
LIN {X 0,Y 192.702,Z 281.984,A -85,B 0,C 180,E1 -21761.481,E2 -21761.481} C_VEL
LIN {X 0,Y 192.74,Z 281.977,A -85,B 0,C 180,E1 -21765.2,E2 -21765.2} C_VEL
LIN {X 0,Y 192.948,Z 281.952,A -85,B 0,C 180,E1 -21769.555,E2 -21769.555} C_VEL
LIN {X 0,Y 192.969,Z 281.949,A -85,B 0,C 180,E1 -21773.715,E2 -21773.715} C_VEL
LIN {X 0,Y 193.229,Z 281.912,A -85,B 0,C 180,E1 -21777.904,E2 -21777.904} C_VEL
LIN {X 0,Y 193.427,Z 281.869,A -85,B 0,C 180,E1 -21779.988,E2 -21779.988} C_VEL
LIN {X 0,Y 192.953,Z 281.935,A -85,B 0,C 180,E1 -21784.165,E2 -21784.165} C_VEL
LIN {X 0,Y 193.017,Z 281.94,A -85,B 0,C 180,E1 -21788.362,E2 -21788.362} C_VEL
LIN {X 0,Y 192.775,Z 281.973,A -85,B 0,C 180,E1 -21792.622,E2 -21792.622} C_VEL
LIN {X 0,Y 192.698,Z 281.983,A -85,B 0,C 180,E1 -21796.95,E2 -21796.95} C_VEL
LIN {X 0,Y 192.562,Z 281.998,A -85,B 0,C 180,E1 -21801.391,E2 -21801.391} C_VEL
LIN {X 0,Y 192.617,Z 281.986,A -85,B 0,C 180,E1 -21804.196,E2 -21804.196} C_VEL
LIN {X 0,Y 192.61,Z 281.992,A -85,B 0,C 180,E1 -21808.873,E2 -21808.873} C_VEL
LIN {X 0,Y 192.567,Z 281.996,A -85,B 0,C 180,E1 -21813.175,E2 -21813.175} C_VEL
LIN {X 0,Y 192.568,Z 281.997,A -85,B 0,C 180,E1 -21818.33,E2 -21818.33} C_VEL
LIN {X 0,Y 192.576,Z 281.996,A -85,B 0,C 180,E1 -21823.124,E2 -21823.124} C_VEL
LIN {X 0,Y 192.574,Z 281.996,A -85,B 0,C 180,E1 -21826.857,E2 -21826.857} C_VEL
LIN {X 0,Y 192.578,Z 282.113,A -85,B 0,C 180,E1 -21829.942,E2 -21829.942} C_VEL
LIN {X 0,Y 193.484,Z 284.685,A -85,B 0,C 180,E1 -21830.333,E2 -21830.333} C_VEL
LIN {X 0,Y 195.34,Z 287.28,A -85,B 0,C 180,E1 -21830.948,E2 -21830.948} C_VEL
LIN {X 0,Y 202.011,Z 299.544,A -85,B 0,C 180,E1 -21833.6,E2 -21833.6} C_VEL
LIN {X 0,Y 206.757,Z 310.349,A -85,B 0,C 180,E1 -21835.92,E2 -21835.92} C_VEL
LIN {X 0,Y 210.179,Z 319.886,A -85,B 0,C 180,E1 -21838.02,E2 -21838.02} C_VEL
LIN {X 0,Y 213.119,Z 329.836,A -85,B 0,C 180,E1 -21840.354,E2 -21840.354} C_VEL
LIN {X 0,Y 216.31,Z 338.1,A -85,B 0,C 180,E1 -21842.624,E2 -21842.624} C_VEL
LIN {X 0,Y 220.686,Z 346.294,A -85,B 0,C 180,E1 -21845.251,E2 -21845.251} C_VEL
LIN {X 0,Y 226.311,Z 354.049,A -85,B 0,C 180,E1 -21848.121,E2 -21848.121} C_VEL
LIN {X 0,Y 233.638,Z 361.573,A -85,B 0,C 180,E1 -21851.315,E2 -21851.315} C_VEL
LIN {X 0,Y 242.993,Z 368.886,A -85,B 0,C 180,E1 -21854.912,E2 -21854.912} C_VEL
LIN {X 0,Y 251.512,Z 374.051,A -85,B 0,C 180,E1 -21857.899,E2 -21857.899} C_VEL
LIN {X 0,Y 259.193,Z 378.098,A -85,B 0,C 180,E1 -21860.637,E2 -21860.637} C_VEL
LIN {X 0,Y 263.767,Z 380.227,A -85,B 0,C 180,E1 -21862.344,E2 -21862.344} C_VEL
LIN {X 0,Y 268.331,Z 382.226,A -85,B 0,C 180,E1 -21864.304,E2 -21864.304} C_VEL
LIN {X 0,Y 270.511,Z 383.213,A -85,B 0,C 180,E1 -21865.53,E2 -21865.53} C_VEL
LIN {X 0,Y 274.198,Z 384.521,A -85,B 0,C 180,E1 -21868.02,E2 -21868.02} C_VEL
LIN {X 0,Y 276.115,Z 384.841,A -85,B 0,C 180,E1 -21870,E2 -21870} C_VEL
LIN {X 0,Y 274.197,Z 384.523,A -85,B 0,C 180,E1 -21871.975,E2 -21871.975} C_VEL
LIN {X 0,Y 270.509,Z 383.212,A -85,B 0,C 180,E1 -21874.47,E2 -21874.47} C_VEL
LIN {X 0,Y 267.587,Z 381.92,A -85,B 0,C 180,E1 -21876.03,E2 -21876.03} C_VEL
LIN {X 0,Y 262.603,Z 379.697,A -85,B 0,C 180,E1 -21878.107,E2 -21878.107} C_VEL
LIN {X 0,Y 256.991,Z 376.978,A -85,B 0,C 180,E1 -21880.173,E2 -21880.173} C_VEL
LIN {X 0,Y 248.743,Z 372.471,A -85,B 0,C 180,E1 -21883.063,E2 -21883.063} C_VEL
LIN {X 0,Y 240.99,Z 367.495,A -85,B 0,C 180,E1 -21885.815,E2 -21885.815} C_VEL
LIN {X 0,Y 233.642,Z 361.564,A -85,B 0,C 180,E1 -21888.688,E2 -21888.688} C_VEL
LIN {X 0,Y 226.295,Z 354.05,A -85,B 0,C 180,E1 -21891.881,E2 -21891.881} C_VEL
LIN {X 0,Y 220.645,Z 346.29,A -85,B 0,C 180,E1 -21894.755,E2 -21894.755} C_VEL
LIN {X 0,Y 216.3,Z 338.132,A -85,B 0,C 180,E1 -21897.37,E2 -21897.37} C_VEL
LIN {X 0,Y 212.782,Z 328.785,A -85,B 0,C 180,E1 -21899.915,E2 -21899.915} C_VEL
LIN {X 0,Y 209.524,Z 317.787,A -85,B 0,C 180,E1 -21902.457,E2 -21902.457} C_VEL
LIN {X 0,Y 204.908,Z 305.821,A -85,B 0,C 180,E1 -21905.053,E2 -21905.053} C_VEL
LIN {X 0,Y 199.946,Z 295.677,A -85,B 0,C 180,E1 -21907.241,E2 -21907.241} C_VEL
LIN {X 0,Y 194.59,Z 286.111,A -85,B 0,C 180,E1 -21909.319,E2 -21909.319} C_VEL
LIN {X 0,Y 193.015,Z 283.725,A -85,B 0,C 180,E1 -21909.87,E2 -21909.87} C_VEL
LIN {X 0,Y 192.557,Z 281.998,A -85,B 0,C 180,E1 -21910.145,E2 -21910.145} C_VEL
LIN {X 0,Y 192.582,Z 281.998,A -85,B 0,C 180,E1 -21913.897,E2 -21913.897} C_VEL
LIN {X 0,Y 192.576,Z 281.996,A -85,B 0,C 180,E1 -21916.876,E2 -21916.876} C_VEL
LIN {X 0,Y 192.568,Z 281.997,A -85,B 0,C 180,E1 -21921.67,E2 -21921.67} C_VEL
LIN {X 0,Y 192.567,Z 281.996,A -85,B 0,C 180,E1 -21926.825,E2 -21926.825} C_VEL
LIN {X 0,Y 192.627,Z 281.99,A -85,B 0,C 180,E1 -21931.702,E2 -21931.702} C_VEL
LIN {X 0,Y 192.651,Z 281.985,A -85,B 0,C 180,E1 -21936.356,E2 -21936.356} C_VEL
LIN {X 0,Y 192.676,Z 281.982,A -85,B 0,C 180,E1 -21941.504,E2 -21941.504} C_VEL
LIN {X 0,Y 192.719,Z 281.972,A -85,B 0,C 180,E1 -21945.224,E2 -21945.224} C_VEL
LIN {X 0,Y 192.934,Z 281.947,A -85,B 0,C 180,E1 -21949.579,E2 -21949.579} C_VEL
LIN {X 0,Y 192.965,Z 281.947,A -85,B 0,C 180,E1 -21953.74,E2 -21953.74} C_VEL
LIN {X 0,Y 193.251,Z 281.88,A -85,B 0,C 180,E1 -21957.928,E2 -21957.928} C_VEL
LIN {X 0,Y 193.427,Z 281.869,A -85,B 0,C 180,E1 -21960.012,E2 -21960.012} C_VEL
LIN {X 0,Y 192.938,Z 281.952,A -85,B 0,C 180,E1 -21964.19,E2 -21964.19} C_VEL
LIN {X 0,Y 193.028,Z 281.942,A -85,B 0,C 180,E1 -21968.386,E2 -21968.386} C_VEL
LIN {X 0,Y 192.793,Z 281.972,A -85,B 0,C 180,E1 -21972.646,E2 -21972.646} C_VEL
LIN {X 0,Y 192.722,Z 281.981,A -85,B 0,C 180,E1 -21976.974,E2 -21976.974} C_VEL
LIN {X 0,Y 192.588,Z 281.996,A -85,B 0,C 180,E1 -21981.415,E2 -21981.415} C_VEL
LIN {X 0,Y 192.637,Z 281.991,A -85,B 0,C 180,E1 -21984.209,E2 -21984.209} C_VEL
LIN {X 0,Y 192.778,Z 283.38,A -85,B 0,C 180,E1 -21988.963,E2 -21988.963} C_VEL
LIN {X 0,Y 192.998,Z 284.9,A -85,B 0,C 180,E1 -21993.121,E2 -21993.121} C_VEL
LIN {X 0,Y 193.261,Z 286.953,A -85,B 0,C 180,E1 -21998.198,E2 -21998.198} C_VEL
LIN {X 0,Y 193.447,Z 288.144,A -85,B 0,C 180,E1 -22000.853,E2 -22000.853} C_VEL
LIN {X 0,Y 193.537,Z 289.47,A -85,B 0,C 180,E1 -22003.64,E2 -22003.64} C_VEL
LIN {X 0,Y 193.451,Z 290.988,A -85,B 0,C 180,E1 -22006.615,E2 -22006.615} C_VEL
LIN {X 0,Y 193.074,Z 292.958,A -85,B 0,C 180,E1 -22010.192,E2 -22010.192} C_VEL
LIN {X 0,Y 194.095,Z 296.37,A -85,B 0,C 180,E1 -22010.708,E2 -22010.708} C_VEL
LIN {X 0,Y 195.094,Z 298.848,A -85,B 0,C 180,E1 -22011.166,E2 -22011.166} C_VEL
LIN {X 0,Y 198.467,Z 308.266,A -85,B 0,C 180,E1 -22012.838,E2 -22012.838} C_VEL
LIN {X 0,Y 201.268,Z 319.599,A -85,B 0,C 180,E1 -22014.869,E2 -22014.869} C_VEL
LIN {X 0,Y 203.035,Z 329.721,A -85,B 0,C 180,E1 -22016.814,E2 -22016.814} C_VEL
LIN {X 0,Y 203.837,Z 337.755,A -85,B 0,C 180,E1 -22018.456,E2 -22018.456} C_VEL
LIN {X 0,Y 204.145,Z 346.755,A -85,B 0,C 180,E1 -22020.484,E2 -22020.484} C_VEL
LIN {X 0,Y 203.861,Z 353.976,A -85,B 0,C 180,E1 -22022.264,E2 -22022.264} C_VEL
LIN {X 0,Y 200.939,Z 363.111,A -85,B 0,C 180,E1 -22024.631,E2 -22024.631} C_VEL
LIN {X 0,Y 198.89,Z 369.314,A -85,B 0,C 180,E1 -22026.577,E2 -22026.577} C_VEL
LIN {X 0,Y 196.691,Z 375.853,A -85,B 0,C 180,E1 -22029.065,E2 -22029.065} C_VEL
LIN {X 0,Y 195.089,Z 380.355,A -85,B 0,C 180,E1 -22031.082,E2 -22031.082} C_VEL
LIN {X 0,Y 193.053,Z 385.845,A -85,B 0,C 180,E1 -22034.156,E2 -22034.156} C_VEL
LIN {X 0,Y 191.662,Z 390.175,A -85,B 0,C 180,E1 -22037.291,E2 -22037.291} C_VEL
LIN {X 0,Y 191.016,Z 392.546,A -85,B 0,C 180,E1 -22039.4,E2 -22039.4} C_VEL
LIN {X 0,Y 190.543,Z 394.349,A -85,B 0,C 180,E1 -22041.516,E2 -22041.516} C_VEL
LIN {X 0,Y 190.115,Z 396.804,A -85,B 0,C 180,E1 -22045.76,E2 -22045.76} C_VEL
LIN {X 0,Y 190.152,Z 397.399,A -85,B 0,C 180,E1 -22047.882,E2 -22047.882} C_VEL
LIN {X 0,Y 190.236,Z 397.557,A -85,B 0,C 180,E1 -22050,E2 -22050} C_VEL
LIN {X 0,Y 190.14,Z 397.012,A -85,B 0,C 180,E1 -22053.5,E2 -22053.5} C_VEL
LIN {X 0,Y 190.24,Z 395.741,A -85,B 0,C 180,E1 -22056.363,E2 -22056.363} C_VEL
LIN {X 0,Y 190.516,Z 394.378,A -85,B 0,C 180,E1 -22058.44,E2 -22058.44} C_VEL
LIN {X 0,Y 190.227,Z 393.045,A -85,B 0,C 180,E1 -22060.168,E2 -22060.168} C_VEL
LIN {X 0,Y 188.194,Z 390.163,A -85,B 0,C 180,E1 -22062.975,E2 -22062.975} C_VEL
LIN {X 0,Y 186.52,Z 386.578,A -85,B 0,C 180,E1 -22065.768,E2 -22065.768} C_VEL
LIN {X 0,Y 186.808,Z 384.126,A -85,B 0,C 180,E1 -22067.423,E2 -22067.423} C_VEL
LIN {X 0,Y 189.124,Z 377.967,A -85,B 0,C 180,E1 -22070.672,E2 -22070.672} C_VEL
LIN {X 0,Y 191.25,Z 372.417,A -85,B 0,C 180,E1 -22073.041,E2 -22073.041} C_VEL
LIN {X 0,Y 193.352,Z 366.168,A -85,B 0,C 180,E1 -22075.282,E2 -22075.282} C_VEL
LIN {X 0,Y 196.314,Z 357.618,A -85,B 0,C 180,E1 -22077.735,E2 -22077.735} C_VEL
LIN {X 0,Y 197.286,Z 353.771,A -85,B 0,C 180,E1 -22078.745,E2 -22078.745} C_VEL
LIN {X 0,Y 197.609,Z 343.353,A -85,B 0,C 180,E1 -22081.381,E2 -22081.381} C_VEL
LIN {X 0,Y 196.885,Z 332.526,A -85,B 0,C 180,E1 -22083.801,E2 -22083.801} C_VEL
LIN {X 0,Y 195.325,Z 322.295,A -85,B 0,C 180,E1 -22085.911,E2 -22085.911} C_VEL
LIN {X 0,Y 193.555,Z 314.3,A -85,B 0,C 180,E1 -22087.483,E2 -22087.483} C_VEL
LIN {X 0,Y 190.173,Z 303.549,A -85,B 0,C 180,E1 -22089.56,E2 -22089.56} C_VEL
LIN {X 0,Y 187.585,Z 296.811,A -85,B 0,C 180,E1 -22090.881,E2 -22090.881} C_VEL
LIN {X 0,Y 186.32,Z 293.755,A -85,B 0,C 180,E1 -22091.44,E2 -22091.44} C_VEL
LIN {X 0,Y 186.169,Z 292.75,A -85,B 0,C 180,E1 -22091.609,E2 -22091.609} C_VEL
LIN {X 0,Y 186.457,Z 290.648,A -85,B 0,C 180,E1 -22095.736,E2 -22095.736} C_VEL
LIN {X 0,Y 186.361,Z 288.639,A -85,B 0,C 180,E1 -22100.113,E2 -22100.113} C_VEL
LIN {X 0,Y 185.996,Z 286.441,A -85,B 0,C 180,E1 -22105.461,E2 -22105.461} C_VEL
LIN {X 0,Y 185.769,Z 284.623,A -85,B 0,C 180,E1 -22110.527,E2 -22110.527} C_VEL
LIN {X 0,Y 185.592,Z 283.08,A -85,B 0,C 180,E1 -22115.371,E2 -22115.371} C_VEL
LIN {X 0,Y 185.54,Z 282.877,A -85,B 0,C 180,E1 -22120.056,E2 -22120.056} C_VEL
LIN {X 0,Y 185.659,Z 282.86,A -85,B 0,C 180,E1 -22122.36,E2 -22122.36} C_VEL
LIN {X 0,Y 185.719,Z 282.851,A -85,B 0,C 180,E1 -22126.864,E2 -22126.864} C_VEL
LIN {X 0,Y 185.977,Z 282.821,A -85,B 0,C 180,E1 -22131.294,E2 -22131.294} C_VEL
LIN {X 0,Y 186.175,Z 282.79,A -85,B 0,C 180,E1 -22137.824,E2 -22137.824} C_VEL
LIN {X 0,Y 186.391,Z 282.744,A -85,B 0,C 180,E1 -22139.987,E2 -22139.987} C_VEL
LIN {X 0,Y 185.9,Z 282.814,A -85,B 0,C 180,E1 -22144.323,E2 -22144.323} C_VEL
LIN {X 0,Y 185.965,Z 282.815,A -85,B 0,C 180,E1 -22148.681,E2 -22148.681} C_VEL
LIN {X 0,Y 185.7,Z 282.851,A -85,B 0,C 180,E1 -22153.111,E2 -22153.111} C_VEL
LIN {X 0,Y 185.635,Z 282.861,A -85,B 0,C 180,E1 -22157.616,E2 -22157.616} C_VEL
LIN {X 0,Y 185.533,Z 282.874,A -85,B 0,C 180,E1 -22162.244,E2 -22162.244} C_VEL
LIN {X 0,Y 185.528,Z 282.876,A -85,B 0,C 180,E1 -22167.021,E2 -22167.021} C_VEL
LIN {X 0,Y 185.55,Z 282.872,A -85,B 0,C 180,E1 -22169.482,E2 -22169.482} C_VEL
LIN {X 0,Y 185.489,Z 282.881,A -85,B 0,C 180,E1 -22174.616,E2 -22174.616} C_VEL
LIN {X 0,Y 185.537,Z 282.874,A -85,B 0,C 180,E1 -22177.303,E2 -22177.303} C_VEL
LIN {X 0,Y 185.528,Z 282.874,A -85,B 0,C 180,E1 -22180.747,E2 -22180.747} C_VEL
LIN {X 0,Y 185.541,Z 282.874,A -85,B 0,C 180,E1 -22186.007,E2 -22186.007} C_VEL
LIN {X 0,Y 185.483,Z 282.885,A -85,B 0,C 180,E1 -22188.109,E2 -22188.109} C_VEL
LIN {X 0,Y 186.499,Z 285.732,A -85,B 0,C 180,E1 -22188.584,E2 -22188.584} C_VEL
LIN {X 0,Y 188.345,Z 288.134,A -85,B 0,C 180,E1 -22189.245,E2 -22189.245} C_VEL
LIN {X 0,Y 194.27,Z 298.68,A -85,B 0,C 180,E1 -22191.762,E2 -22191.762} C_VEL
LIN {X 0,Y 199.175,Z 309.262,A -85,B 0,C 180,E1 -22194.224,E2 -22194.224} C_VEL
LIN {X 0,Y 203.004,Z 319.372,A -85,B 0,C 180,E1 -22196.611,E2 -22196.611} C_VEL
LIN {X 0,Y 205.532,Z 328.076,A -85,B 0,C 180,E1 -22198.716,E2 -22198.716} C_VEL
LIN {X 0,Y 208.383,Z 337.318,A -85,B 0,C 180,E1 -22201.239,E2 -22201.239} C_VEL
LIN {X 0,Y 212.018,Z 345.421,A -85,B 0,C 180,E1 -22203.852,E2 -22203.852} C_VEL
LIN {X 0,Y 216.514,Z 352.691,A -85,B 0,C 180,E1 -22206.558,E2 -22206.558} C_VEL
LIN {X 0,Y 221.548,Z 358.802,A -85,B 0,C 180,E1 -22209.135,E2 -22209.135} C_VEL
LIN {X 0,Y 228.638,Z 365.391,A -85,B 0,C 180,E1 -22212.299,E2 -22212.299} C_VEL
LIN {X 0,Y 236.121,Z 370.801,A -85,B 0,C 180,E1 -22215.261,E2 -22215.261} C_VEL
LIN {X 0,Y 244.871,Z 375.762,A -85,B 0,C 180,E1 -22218.41,E2 -22218.41} C_VEL
LIN {X 0,Y 252.646,Z 379.45,A -85,B 0,C 180,E1 -22221.2,E2 -22221.2} C_VEL
LIN {X 0,Y 259.234,Z 382.151,A -85,B 0,C 180,E1 -22223.775,E2 -22223.775} C_VEL
LIN {X 0,Y 262.706,Z 383.426,A -85,B 0,C 180,E1 -22225.397,E2 -22225.397} C_VEL
LIN {X 0,Y 265.21,Z 384.361,A -85,B 0,C 180,E1 -22226.962,E2 -22226.962} C_VEL
LIN {X 0,Y 267.469,Z 384.884,A -85,B 0,C 180,E1 -22228.494,E2 -22228.494} C_VEL
LIN {X 0,Y 268.886,Z 385.036,A -85,B 0,C 180,E1 -22230,E2 -22230} C_VEL
LIN {X 0,Y 267.129,Z 384.814,A -85,B 0,C 180,E1 -22231.739,E2 -22231.739} C_VEL
LIN {X 0,Y 265.206,Z 384.361,A -85,B 0,C 180,E1 -22233.038,E2 -22233.038} C_VEL
LIN {X 0,Y 262.708,Z 383.425,A -85,B 0,C 180,E1 -22234.603,E2 -22234.603} C_VEL
LIN {X 0,Y 259.24,Z 382.151,A -85,B 0,C 180,E1 -22236.225,E2 -22236.225} C_VEL
LIN {X 0,Y 255.047,Z 380.469,A -85,B 0,C 180,E1 -22237.919,E2 -22237.919} C_VEL
LIN {X 0,Y 247.595,Z 377.129,A -85,B 0,C 180,E1 -22240.633,E2 -22240.633} C_VEL
LIN {X 0,Y 238.744,Z 372.429,A -85,B 0,C 180,E1 -22243.784,E2 -22243.784} C_VEL
LIN {X 0,Y 231.086,Z 367.306,A -85,B 0,C 180,E1 -22246.71,E2 -22246.71} C_VEL
LIN {X 0,Y 223.95,Z 361.242,A -85,B 0,C 180,E1 -22249.743,E2 -22249.743} C_VEL
LIN {X 0,Y 217.678,Z 354.298,A -85,B 0,C 180,E1 -22252.794,E2 -22252.794} C_VEL
LIN {X 0,Y 213.193,Z 347.618,A -85,B 0,C 180,E1 -22255.375,E2 -22255.375} C_VEL
LIN {X 0,Y 209.305,Z 339.679,A -85,B 0,C 180,E1 -22258.039,E2 -22258.039} C_VEL
LIN {X 0,Y 206.449,Z 331.525,A -85,B 0,C 180,E1 -22260.39,E2 -22260.39} C_VEL
LIN {X 0,Y 203.745,Z 321.807,A -85,B 0,C 180,E1 -22262.803,E2 -22262.803} C_VEL
LIN {X 0,Y 200.91,Z 313.683,A -85,B 0,C 180,E1 -22264.733,E2 -22264.733} C_VEL
LIN {X 0,Y 197.308,Z 304.935,A -85,B 0,C 180,E1 -22266.757,E2 -22266.757} C_VEL
LIN {X 0,Y 192.185,Z 294.776,A -85,B 0,C 180,E1 -22269.133,E2 -22269.133} C_VEL
LIN {X 0,Y 188.247,Z 287.958,A -85,B 0,C 180,E1 -22270.794,E2 -22270.794} C_VEL
LIN {X 0,Y 186.031,Z 284.826,A -85,B 0,C 180,E1 -22271.63,E2 -22271.63} C_VEL
LIN {X 0,Y 185.496,Z 282.879,A -85,B 0,C 180,E1 -22271.971,E2 -22271.971} C_VEL
LIN {X 0,Y 185.542,Z 282.875,A -85,B 0,C 180,E1 -22276.027,E2 -22276.027} C_VEL
LIN {X 0,Y 185.508,Z 282.877,A -85,B 0,C 180,E1 -22279.925,E2 -22279.925} C_VEL
LIN {X 0,Y 185.528,Z 282.875,A -85,B 0,C 180,E1 -22282.711,E2 -22282.711} C_VEL
LIN {X 0,Y 185.508,Z 282.877,A -85,B 0,C 180,E1 -22287.985,E2 -22287.985} C_VEL
LIN {X 0,Y 185.553,Z 282.872,A -85,B 0,C 180,E1 -22290.59,E2 -22290.59} C_VEL
LIN {X 0,Y 185.558,Z 282.864,A -85,B 0,C 180,E1 -22295.394,E2 -22295.394} C_VEL
LIN {X 0,Y 185.607,Z 282.859,A -85,B 0,C 180,E1 -22301.192,E2 -22301.192} C_VEL
LIN {X 0,Y 185.649,Z 282.854,A -85,B 0,C 180,E1 -22304.647,E2 -22304.647} C_VEL
LIN {X 0,Y 185.876,Z 282.826,A -85,B 0,C 180,E1 -22309.432,E2 -22309.432} C_VEL
LIN {X 0,Y 185.929,Z 282.824,A -85,B 0,C 180,E1 -22313.502,E2 -22313.502} C_VEL
LIN {X 0,Y 186.195,Z 282.758,A -85,B 0,C 180,E1 -22317.85,E2 -22317.85} C_VEL
LIN {X 0,Y 186.391,Z 282.744,A -85,B 0,C 180,E1 -22320.013,E2 -22320.013} C_VEL
LIN {X 0,Y 185.887,Z 282.83,A -85,B 0,C 180,E1 -22324.349,E2 -22324.349} C_VEL
LIN {X 0,Y 185.977,Z 282.82,A -85,B 0,C 180,E1 -22328.706,E2 -22328.706} C_VEL
LIN {X 0,Y 185.719,Z 282.853,A -85,B 0,C 180,E1 -22333.136,E2 -22333.136} C_VEL
LIN {X 0,Y 185.659,Z 282.86,A -85,B 0,C 180,E1 -22337.64,E2 -22337.64} C_VEL
LIN {X 0,Y 185.558,Z 282.873,A -85,B 0,C 180,E1 -22342.268,E2 -22342.268} C_VEL
LIN {X 0,Y 185.591,Z 283.086,A -85,B 0,C 180,E1 -22344.658,E2 -22344.658} C_VEL
LIN {X 0,Y 185.779,Z 284.643,A -85,B 0,C 180,E1 -22349.534,E2 -22349.534} C_VEL
LIN {X 0,Y 185.996,Z 286.44,A -85,B 0,C 180,E1 -22354.539,E2 -22354.539} C_VEL
LIN {X 0,Y 186.197,Z 287.659,A -85,B 0,C 180,E1 -22357.569,E2 -22357.569} C_VEL
LIN {X 0,Y 186.405,Z 289.166,A -85,B 0,C 180,E1 -22361.058,E2 -22361.058} C_VEL
LIN {X 0,Y 186.419,Z 291.379,A -85,B 0,C 180,E1 -22365.764,E2 -22365.764} C_VEL
LIN {X 0,Y 186.187,Z 292.924,A -85,B 0,C 180,E1 -22368.465,E2 -22368.465} C_VEL
LIN {X 0,Y 187.214,Z 296.101,A -85,B 0,C 180,E1 -22368.961,E2 -22368.961} C_VEL
LIN {X 0,Y 188.331,Z 298.534,A -85,B 0,C 180,E1 -22369.482,E2 -22369.482} C_VEL
LIN {X 0,Y 191.616,Z 307.652,A -85,B 0,C 180,E1 -22371.22,E2 -22371.22} C_VEL
LIN {X 0,Y 194.39,Z 317.62,A -85,B 0,C 180,E1 -22373.152,E2 -22373.152} C_VEL
LIN {X 0,Y 196.381,Z 328.863,A -85,B 0,C 180,E1 -22375.414,E2 -22375.414} C_VEL
LIN {X 0,Y 197.324,Z 337.842,A -85,B 0,C 180,E1 -22377.354,E2 -22377.354} C_VEL
LIN {X 0,Y 197.626,Z 347.108,A -85,B 0,C 180,E1 -22379.552,E2 -22379.552} C_VEL
LIN {X 0,Y 197.321,Z 353.772,A -85,B 0,C 180,E1 -22381.261,E2 -22381.261} C_VEL
LIN {X 0,Y 196.338,Z 357.619,A -85,B 0,C 180,E1 -22382.268,E2 -22382.268} C_VEL
LIN {X 0,Y 193.42,Z 366.17,A -85,B 0,C 180,E1 -22384.727,E2 -22384.727} C_VEL
LIN {X 0,Y 190.597,Z 374.307,A -85,B 0,C 180,E1 -22387.697,E2 -22387.697} C_VEL
LIN {X 0,Y 188.337,Z 380.159,A -85,B 0,C 180,E1 -22390.377,E2 -22390.377} C_VEL
LIN {X 0,Y 186.206,Z 385.65,A -85,B 0,C 180,E1 -22393.557,E2 -22393.557} C_VEL
LIN {X 0,Y 184.702,Z 389.979,A -85,B 0,C 180,E1 -22396.803,E2 -22396.803} C_VEL
LIN {X 0,Y 183.999,Z 392.35,A -85,B 0,C 180,E1 -22398.99,E2 -22398.99} C_VEL
LIN {X 0,Y 183.516,Z 394.154,A -85,B 0,C 180,E1 -22401.189,E2 -22401.189} C_VEL
LIN {X 0,Y 183.044,Z 396.61,A -85,B 0,C 180,E1 -22405.596,E2 -22405.596} C_VEL
LIN {X 0,Y 183.07,Z 397.204,A -85,B 0,C 180,E1 -22407.8,E2 -22407.8} C_VEL
LIN {X 0,Y 183.144,Z 397.362,A -85,B 0,C 180,E1 -22410,E2 -22410} C_VEL
LIN {X 0,Y 183.042,Z 396.937,A -85,B 0,C 180,E1 -22413.191,E2 -22413.191} C_VEL
LIN {X 0,Y 183.162,Z 395.545,A -85,B 0,C 180,E1 -22416.61,E2 -22416.61} C_VEL
LIN {X 0,Y 183.476,Z 394.153,A -85,B 0,C 180,E1 -22418.813,E2 -22418.813} C_VEL
LIN {X 0,Y 184.333,Z 391.198,A -85,B 0,C 180,E1 -22422.104,E2 -22422.104} C_VEL
LIN {X 0,Y 185.591,Z 387.203,A -85,B 0,C 180,E1 -22425.371,E2 -22425.371} C_VEL
LIN {X 0,Y 186.808,Z 384.126,A -85,B 0,C 180,E1 -22427.423,E2 -22427.423} C_VEL
LIN {X 0,Y 187.228,Z 381.474,A -85,B 0,C 180,E1 -22429.035,E2 -22429.035} C_VEL
LIN {X 0,Y 186.33,Z 376.606,A -85,B 0,C 180,E1 -22431.674,E2 -22431.674} C_VEL
LIN {X 0,Y 185.629,Z 371.21,A -85,B 0,C 180,E1 -22434.235,E2 -22434.235} C_VEL
LIN {X 0,Y 186.351,Z 367.589,A -85,B 0,C 180,E1 -22435.68,E2 -22435.68} C_VEL
LIN {X 0,Y 189.393,Z 359.342,A -85,B 0,C 180,E1 -22438.237,E2 -22438.237} C_VEL
LIN {X 0,Y 190.569,Z 355.5,A -85,B 0,C 180,E1 -22439.251,E2 -22439.251} C_VEL
LIN {X 0,Y 191.147,Z 346.955,A -85,B 0,C 180,E1 -22441.582,E2 -22441.582} C_VEL
LIN {X 0,Y 190.77,Z 336.631,A -85,B 0,C 180,E1 -22444.149,E2 -22444.149} C_VEL
LIN {X 0,Y 189.243,Z 324.295,A -85,B 0,C 180,E1 -22446.893,E2 -22446.893} C_VEL
LIN {X 0,Y 187.265,Z 315.088,A -85,B 0,C 180,E1 -22448.84,E2 -22448.84} C_VEL
LIN {X 0,Y 183.875,Z 304.253,A -85,B 0,C 180,E1 -22451.105,E2 -22451.105} C_VEL
LIN {X 0,Y 180.925,Z 296.89,A -85,B 0,C 180,E1 -22452.701,E2 -22452.701} C_VEL
LIN {X 0,Y 179.56,Z 293.976,A -85,B 0,C 180,E1 -22453.34,E2 -22453.34} C_VEL
LIN {X 0,Y 179.293,Z 292.54,A -85,B 0,C 180,E1 -22453.548,E2 -22453.548} C_VEL
LIN {X 0,Y 179.376,Z 290.399,A -85,B 0,C 180,E1 -22458.222,E2 -22458.222} C_VEL
LIN {X 0,Y 179.199,Z 288.943,A -85,B 0,C 180,E1 -22461.662,E2 -22461.662} C_VEL
LIN {X 0,Y 178.915,Z 287.011,A -85,B 0,C 180,E1 -22466.624,E2 -22466.624} C_VEL
LIN {X 0,Y 178.663,Z 285.265,A -85,B 0,C 180,E1 -22471.82,E2 -22471.82} C_VEL
LIN {X 0,Y 178.486,Z 283.802,A -85,B 0,C 180,E1 -22476.799,E2 -22476.799} C_VEL
LIN {X 0,Y 178.615,Z 283.739,A -85,B 0,C 180,E1 -22481.64,E2 -22481.64} C_VEL
LIN {X 0,Y 178.646,Z 283.732,A -85,B 0,C 180,E1 -22486.334,E2 -22486.334} C_VEL
LIN {X 0,Y 178.908,Z 283.7,A -85,B 0,C 180,E1 -22490.947,E2 -22490.947} C_VEL
LIN {X 0,Y 179.123,Z 283.669,A -85,B 0,C 180,E1 -22497.738,E2 -22497.738} C_VEL
LIN {X 0,Y 179.354,Z 283.618,A -85,B 0,C 180,E1 -22499.987,E2 -22499.987} C_VEL
LIN {X 0,Y 178.847,Z 283.694,A -85,B 0,C 180,E1 -22504.494,E2 -22504.494} C_VEL
LIN {X 0,Y 178.895,Z 283.694,A -85,B 0,C 180,E1 -22509.027,E2 -22509.027} C_VEL
LIN {X 0,Y 178.627,Z 283.73,A -85,B 0,C 180,E1 -22513.64,E2 -22513.64} C_VEL
LIN {X 0,Y 178.535,Z 283.738,A -85,B 0,C 180,E1 -22519.138,E2 -22519.138} C_VEL
LIN {X 0,Y 178.497,Z 283.743,A -85,B 0,C 180,E1 -22525.101,E2 -22525.101} C_VEL
LIN {X 0,Y 178.493,Z 283.752,A -85,B 0,C 180,E1 -22529.979,E2 -22529.979} C_VEL
LIN {X 0,Y 178.453,Z 283.756,A -85,B 0,C 180,E1 -22534.206,E2 -22534.206} C_VEL
LIN {X 0,Y 178.44,Z 283.758,A -85,B 0,C 180,E1 -22539.043,E2 -22539.043} C_VEL
LIN {X 0,Y 178.468,Z 283.755,A -85,B 0,C 180,E1 -22542.004,E2 -22542.004} C_VEL
LIN {X 0,Y 178.507,Z 283.767,A -85,B 0,C 180,E1 -22546.113,E2 -22546.113} C_VEL
LIN {X 0,Y 179.361,Z 286.348,A -85,B 0,C 180,E1 -22546.566,E2 -22546.566} C_VEL
LIN {X 0,Y 181.378,Z 289.131,A -85,B 0,C 180,E1 -22547.386,E2 -22547.386} C_VEL
LIN {X 0,Y 183.456,Z 292.486,A -85,B 0,C 180,E1 -22548.34,E2 -22548.34} C_VEL
LIN {X 0,Y 188.192,Z 301.169,A -85,B 0,C 180,E1 -22550.591,E2 -22550.591} C_VEL
LIN {X 0,Y 192.474,Z 310.236,A -85,B 0,C 180,E1 -22552.897,E2 -22552.897} C_VEL
LIN {X 0,Y 196.242,Z 320.262,A -85,B 0,C 180,E1 -22555.43,E2 -22555.43} C_VEL
LIN {X 0,Y 198.736,Z 328.866,A -85,B 0,C 180,E1 -22557.648,E2 -22557.648} C_VEL
LIN {X 0,Y 201.25,Z 338.122,A -85,B 0,C 180,E1 -22560.27,E2 -22560.27} C_VEL
LIN {X 0,Y 204.247,Z 345.711,A -85,B 0,C 180,E1 -22562.794,E2 -22562.794} C_VEL
LIN {X 0,Y 208.302,Z 353.018,A -85,B 0,C 180,E1 -22565.604,E2 -22565.604} C_VEL
LIN {X 0,Y 212.256,Z 358.46,A -85,B 0,C 180,E1 -22567.95,E2 -22567.95} C_VEL
LIN {X 0,Y 218.89,Z 365.174,A -85,B 0,C 180,E1 -22571.273,E2 -22571.273} C_VEL
LIN {X 0,Y 226.144,Z 370.682,A -85,B 0,C 180,E1 -22574.4,E2 -22574.4} C_VEL
LIN {X 0,Y 235.356,Z 376.026,A -85,B 0,C 180,E1 -22577.935,E2 -22577.935} C_VEL
LIN {X 0,Y 242.279,Z 379.177,A -85,B 0,C 180,E1 -22580.414,E2 -22580.414} C_VEL
LIN {X 0,Y 248.027,Z 381.451,A -85,B 0,C 180,E1 -22582.533,E2 -22582.533} C_VEL
LIN {X 0,Y 254.752,Z 383.643,A -85,B 0,C 180,E1 -22585.253,E2 -22585.253} C_VEL
LIN {X 0,Y 257.564,Z 384.573,A -85,B 0,C 180,E1 -22586.872,E2 -22586.872} C_VEL
LIN {X 0,Y 260.066,Z 385.106,A -85,B 0,C 180,E1 -22588.513,E2 -22588.513} C_VEL
LIN {X 0,Y 261.627,Z 385.231,A -85,B 0,C 180,E1 -22590,E2 -22590} C_VEL
LIN {X 0,Y 259.959,Z 385.089,A -85,B 0,C 180,E1 -22591.549,E2 -22591.549} C_VEL
LIN {X 0,Y 257.563,Z 384.572,A -85,B 0,C 180,E1 -22593.128,E2 -22593.128} C_VEL
LIN {X 0,Y 253.955,Z 383.413,A -85,B 0,C 180,E1 -22595.095,E2 -22595.095} C_VEL
LIN {X 0,Y 248.037,Z 381.429,A -85,B 0,C 180,E1 -22597.485,E2 -22597.485} C_VEL
LIN {X 0,Y 240.946,Z 378.596,A -85,B 0,C 180,E1 -22600.079,E2 -22600.079} C_VEL
LIN {X 0,Y 231.309,Z 373.888,A -85,B 0,C 180,E1 -22603.581,E2 -22603.581} C_VEL
LIN {X 0,Y 223.33,Z 368.758,A -85,B 0,C 180,E1 -22606.765,E2 -22606.765} C_VEL
LIN {X 0,Y 216.595,Z 363.084,A -85,B 0,C 180,E1 -22609.825,E2 -22609.825} C_VEL
LIN {X 0,Y 210.229,Z 355.861,A -85,B 0,C 180,E1 -22613.211,E2 -22613.211} C_VEL
LIN {X 0,Y 205.58,Z 348.422,A -85,B 0,C 180,E1 -22616.218,E2 -22616.218} C_VEL
LIN {X 0,Y 202.361,Z 341.201,A -85,B 0,C 180,E1 -22618.758,E2 -22618.758} C_VEL
LIN {X 0,Y 199.632,Z 332.332,A -85,B 0,C 180,E1 -22621.412,E2 -22621.412} C_VEL
LIN {X 0,Y 197.105,Z 322.943,A -85,B 0,C 180,E1 -22623.879,E2 -22623.879} C_VEL
LIN {X 0,Y 193.827,Z 313.63,A -85,B 0,C 180,E1 -22626.243,E2 -22626.243} C_VEL
LIN {X 0,Y 189.994,Z 304.838,A -85,B 0,C 180,E1 -22628.468,E2 -22628.468} C_VEL
LIN {X 0,Y 185.364,Z 295.867,A -85,B 0,C 180,E1 -22630.781,E2 -22630.781} C_VEL
LIN {X 0,Y 182.461,Z 291.233,A -85,B 0,C 180,E1 -22632.076,E2 -22632.076} C_VEL
LIN {X 0,Y 180.694,Z 288.042,A -85,B 0,C 180,E1 -22632.911,E2 -22632.911} C_VEL
LIN {X 0,Y 179.096,Z 285.819,A -85,B 0,C 180,E1 -22633.575,E2 -22633.575} C_VEL
LIN {X 0,Y 178.495,Z 283.752,A -85,B 0,C 180,E1 -22633.985,E2 -22633.985} C_VEL
LIN {X 0,Y 178.469,Z 283.755,A -85,B 0,C 180,E1 -22638.434,E2 -22638.434} C_VEL
LIN {X 0,Y 178.428,Z 283.758,A -85,B 0,C 180,E1 -22643.803,E2 -22643.803} C_VEL
LIN {X 0,Y 178.459,Z 283.753,A -85,B 0,C 180,E1 -22646.559,E2 -22646.559} C_VEL
LIN {X 0,Y 178.493,Z 283.752,A -85,B 0,C 180,E1 -22650.021,E2 -22650.021} C_VEL
LIN {X 0,Y 178.497,Z 283.743,A -85,B 0,C 180,E1 -22654.899,E2 -22654.899} C_VEL
LIN {X 0,Y 178.589,Z 283.737,A -85,B 0,C 180,E1 -22661.665,E2 -22661.665} C_VEL
LIN {X 0,Y 178.627,Z 283.73,A -85,B 0,C 180,E1 -22666.36,E2 -22666.36} C_VEL
LIN {X 0,Y 178.895,Z 283.694,A -85,B 0,C 180,E1 -22670.973,E2 -22670.973} C_VEL
LIN {X 0,Y 179.14,Z 283.635,A -85,B 0,C 180,E1 -22677.765,E2 -22677.765} C_VEL
LIN {X 0,Y 179.354,Z 283.618,A -85,B 0,C 180,E1 -22680.013,E2 -22680.013} C_VEL
LIN {X 0,Y 178.898,Z 283.701,A -85,B 0,C 180,E1 -22686.781,E2 -22686.781} C_VEL
LIN {X 0,Y 178.837,Z 283.71,A -85,B 0,C 180,E1 -22690.754,E2 -22690.754} C_VEL
LIN {X 0,Y 178.594,Z 283.741,A -85,B 0,C 180,E1 -22696.002,E2 -22696.002} C_VEL
LIN {X 0,Y 178.562,Z 283.743,A -85,B 0,C 180,E1 -22699.163,E2 -22699.163} C_VEL
LIN {X 0,Y 178.486,Z 283.801,A -85,B 0,C 180,E1 -22703.201,E2 -22703.201} C_VEL
LIN {X 0,Y 178.664,Z 285.263,A -85,B 0,C 180,E1 -22708.18,E2 -22708.18} C_VEL
LIN {X 0,Y 178.918,Z 287.027,A -85,B 0,C 180,E1 -22713.376,E2 -22713.376} C_VEL
LIN {X 0,Y 179.214,Z 289.177,A -85,B 0,C 180,E1 -22718.876,E2 -22718.876} C_VEL
LIN {X 0,Y 179.371,Z 290.453,A -85,B 0,C 180,E1 -22721.89,E2 -22721.89} C_VEL
LIN {X 0,Y 179.29,Z 292.56,A -85,B 0,C 180,E1 -22726.452,E2 -22726.452} C_VEL
LIN {X 0,Y 180.281,Z 295.784,A -85,B 0,C 180,E1 -22727.008,E2 -22727.008} C_VEL
LIN {X 0,Y 181.568,Z 298.336,A -85,B 0,C 180,E1 -22727.638,E2 -22727.638} C_VEL
LIN {X 0,Y 184.473,Z 305.593,A -85,B 0,C 180,E1 -22729.193,E2 -22729.193} C_VEL
LIN {X 0,Y 188.005,Z 317.748,A -85,B 0,C 180,E1 -22731.738,E2 -22731.738} C_VEL
LIN {X 0,Y 189.892,Z 328.551,A -85,B 0,C 180,E1 -22734.034,E2 -22734.034} C_VEL
LIN {X 0,Y 190.873,Z 337.924,A -85,B 0,C 180,E1 -22736.173,E2 -22736.173} C_VEL
LIN {X 0,Y 191.1,Z 346.951,A -85,B 0,C 180,E1 -22738.409,E2 -22738.409} C_VEL
LIN {X 0,Y 190.826,Z 353.568,A -85,B 0,C 180,E1 -22740.186,E2 -22740.186} C_VEL
LIN {X 0,Y 190.058,Z 357.424,A -85,B 0,C 180,E1 -22741.269,E2 -22741.269} C_VEL
LIN {X 0,Y 186.979,Z 365.974,A -85,B 0,C 180,E1 -22743.792,E2 -22743.792} C_VEL
LIN {X 0,Y 183.9,Z 374.382,A -85,B 0,C 180,E1 -22746.978,E2 -22746.978} C_VEL
LIN {X 0,Y 181.611,Z 379.962,A -85,B 0,C 180,E1 -22749.618,E2 -22749.618} C_VEL
LIN {X 0,Y 179.386,Z 385.455,A -85,B 0,C 180,E1 -22752.913,E2 -22752.913} C_VEL
LIN {X 0,Y 177.766,Z 389.783,A -85,B 0,C 180,E1 -22756.278,E2 -22756.278} C_VEL
LIN {X 0,Y 177.008,Z 392.154,A -85,B 0,C 180,E1 -22758.55,E2 -22758.55} C_VEL
LIN {X 0,Y 176.478,Z 393.959,A -85,B 0,C 180,E1 -22760.834,E2 -22760.834} C_VEL
LIN {X 0,Y 175.965,Z 396.415,A -85,B 0,C 180,E1 -22765.418,E2 -22765.418} C_VEL
LIN {X 0,Y 175.979,Z 397.01,A -85,B 0,C 180,E1 -22767.711,E2 -22767.711} C_VEL
LIN {X 0,Y 176.054,Z 397.168,A -85,B 0,C 180,E1 -22770,E2 -22770} C_VEL
LIN {X 0,Y 175.959,Z 396.846,A -85,B 0,C 180,E1 -22772.921,E2 -22772.921} C_VEL
LIN {X 0,Y 175.975,Z 396.415,A -85,B 0,C 180,E1 -22774.581,E2 -22774.581} C_VEL
LIN {X 0,Y 176.447,Z 393.958,A -85,B 0,C 180,E1 -22779.167,E2 -22779.167} C_VEL
LIN {X 0,Y 177.36,Z 391.002,A -85,B 0,C 180,E1 -22782.588,E2 -22782.588} C_VEL
LIN {X 0,Y 178.724,Z 387.008,A -85,B 0,C 180,E1 -22785.977,E2 -22785.977} C_VEL
LIN {X 0,Y 180.854,Z 381.88,A -85,B 0,C 180,E1 -22789.287,E2 -22789.287} C_VEL
LIN {X 0,Y 182.992,Z 376.618,A -85,B 0,C 180,E1 -22791.99,E2 -22791.99} C_VEL
LIN {X 0,Y 185.342,Z 370.298,A -85,B 0,C 180,E1 -22794.652,E2 -22794.652} C_VEL
LIN {X 0,Y 186.351,Z 367.589,A -85,B 0,C 180,E1 -22795.68,E2 -22795.68} C_VEL
LIN {X 0,Y 187.102,Z 363.85,A -85,B 0,C 180,E1 -22797.07,E2 -22797.07} C_VEL
LIN {X 0,Y 186.888,Z 360.008,A -85,B 0,C 180,E1 -22798.465,E2 -22798.465} C_VEL
LIN {X 0,Y 185.274,Z 352.091,A -85,B 0,C 180,E1 -22801.212,E2 -22801.212} C_VEL
LIN {X 0,Y 184.671,Z 346.255,A -85,B 0,C 180,E1 -22802.964,E2 -22802.964} C_VEL
LIN {X 0,Y 184.375,Z 336.251,A -85,B 0,C 180,E1 -22805.549,E2 -22805.549} C_VEL
LIN {X 0,Y 183.087,Z 325.614,A -85,B 0,C 180,E1 -22808.084,E2 -22808.084} C_VEL
LIN {X 0,Y 180.625,Z 314.321,A -85,B 0,C 180,E1 -22810.632,E2 -22810.632} C_VEL
LIN {X 0,Y 177.584,Z 304.922,A -85,B 0,C 180,E1 -22812.801,E2 -22812.801} C_VEL
LIN {X 0,Y 175.868,Z 300.883,A -85,B 0,C 180,E1 -22813.767,E2 -22813.767} C_VEL
LIN {X 0,Y 174.317,Z 297.01,A -85,B 0,C 180,E1 -22814.696,E2 -22814.696} C_VEL
LIN {X 0,Y 172.653,Z 293.963,A -85,B 0,C 180,E1 -22815.524,E2 -22815.524} C_VEL
LIN {X 0,Y 172.302,Z 292.278,A -85,B 0,C 180,E1 -22815.839,E2 -22815.839} C_VEL
LIN {X 0,Y 172.201,Z 290.213,A -85,B 0,C 180,E1 -22820.844,E2 -22820.844} C_VEL
LIN {X 0,Y 171.963,Z 288.612,A -85,B 0,C 180,E1 -22825.084,E2 -22825.084} C_VEL
LIN {X 0,Y 171.682,Z 286.719,A -85,B 0,C 180,E1 -22830.565,E2 -22830.565} C_VEL
LIN {X 0,Y 171.488,Z 285.192,A -85,B 0,C 180,E1 -22835.793,E2 -22835.793} C_VEL
LIN {X 0,Y 171.43,Z 284.635,A -85,B 0,C 180,E1 -22838.335,E2 -22838.335} C_VEL
LIN {X 0,Y 171.515,Z 284.623,A -85,B 0,C 180,E1 -22840.851,E2 -22840.851} C_VEL
LIN {X 0,Y 171.561,Z 284.616,A -85,B 0,C 180,E1 -22845.758,E2 -22845.758} C_VEL
LIN {X 0,Y 171.846,Z 284.579,A -85,B 0,C 180,E1 -22850.571,E2 -22850.571} C_VEL
LIN {X 0,Y 171.786,Z 284.588,A -85,B 0,C 180,E1 -22855.293,E2 -22855.293} C_VEL
LIN {X 0,Y 172.318,Z 284.493,A -85,B 0,C 180,E1 -22859.986,E2 -22859.986} C_VEL
LIN {X 0,Y 171.796,Z 284.573,A -85,B 0,C 180,E1 -22864.679,E2 -22864.679} C_VEL
LIN {X 0,Y 171.833,Z 284.572,A -85,B 0,C 180,E1 -22869.401,E2 -22869.401} C_VEL
LIN {X 0,Y 171.541,Z 284.61,A -85,B 0,C 180,E1 -22874.215,E2 -22874.215} C_VEL
LIN {X 0,Y 171.46,Z 284.618,A -85,B 0,C 180,E1 -22879.486,E2 -22879.486} C_VEL
LIN {X 0,Y 171.433,Z 284.624,A -85,B 0,C 180,E1 -22885.594,E2 -22885.594} C_VEL
LIN {X 0,Y 171.41,Z 284.633,A -85,B 0,C 180,E1 -22890.571,E2 -22890.571} C_VEL
LIN {X 0,Y 171.372,Z 284.638,A -85,B 0,C 180,E1 -22895.02,E2 -22895.02} C_VEL
LIN {X 0,Y 171.395,Z 284.636,A -85,B 0,C 180,E1 -22898.824,E2 -22898.824} C_VEL
LIN {X 0,Y 171.395,Z 284.636,A -85,B 0,C 180,E1 -22903.805,E2 -22903.805} C_VEL
LIN {X 0,Y 172.395,Z 287.431,A -85,B 0,C 180,E1 -22904.396,E2 -22904.396} C_VEL
LIN {X 0,Y 174.451,Z 289.94,A -85,B 0,C 180,E1 -22905.316,E2 -22905.316} C_VEL
LIN {X 0,Y 176.378,Z 293.256,A -85,B 0,C 180,E1 -22906.318,E2 -22906.318} C_VEL
LIN {X 0,Y 181.116,Z 301.41,A -85,B 0,C 180,E1 -22908.727,E2 -22908.727} C_VEL
LIN {X 0,Y 185.821,Z 311.375,A -85,B 0,C 180,E1 -22911.49,E2 -22911.49} C_VEL
LIN {X 0,Y 189.171,Z 320.189,A -85,B 0,C 180,E1 -22913.88,E2 -22913.88} C_VEL
LIN {X 0,Y 191.801,Z 328.684,A -85,B 0,C 180,E1 -22916.231,E2 -22916.231} C_VEL
LIN {X 0,Y 194.238,Z 338.706,A -85,B 0,C 180,E1 -22919.181,E2 -22919.181} C_VEL
LIN {X 0,Y 196.682,Z 345.97,A -85,B 0,C 180,E1 -22921.665,E2 -22921.665} C_VEL
LIN {X 0,Y 200.151,Z 353.214,A -85,B 0,C 180,E1 -22924.525,E2 -22924.525} C_VEL
LIN {X 0,Y 205.176,Z 360.504,A -85,B 0,C 180,E1 -22927.866,E2 -22927.866} C_VEL
LIN {X 0,Y 211.48,Z 366.838,A -85,B 0,C 180,E1 -22931.237,E2 -22931.237} C_VEL
LIN {X 0,Y 218.702,Z 372.23,A -85,B 0,C 180,E1 -22934.537,E2 -22934.537} C_VEL
LIN {X 0,Y 229.283,Z 377.933,A -85,B 0,C 180,E1 -22938.703,E2 -22938.703} C_VEL
LIN {X 0,Y 236.911,Z 380.972,A -85,B 0,C 180,E1 -22941.47,E2 -22941.47} C_VEL
LIN {X 0,Y 241.924,Z 382.631,A -85,B 0,C 180,E1 -22943.327,E2 -22943.327} C_VEL
LIN {X 0,Y 246.76,Z 383.99,A -85,B 0,C 180,E1 -22945.281,E2 -22945.281} C_VEL
LIN {X 0,Y 249.772,Z 384.788,A -85,B 0,C 180,E1 -22946.774,E2 -22946.774} C_VEL
LIN {X 0,Y 253.007,Z 385.374,A -85,B 0,C 180,E1 -22948.799,E2 -22948.799} C_VEL
LIN {X 0,Y 254.326,Z 385.428,A -85,B 0,C 180,E1 -22950,E2 -22950} C_VEL
LIN {X 0,Y 252.378,Z 385.296,A -85,B 0,C 180,E1 -22951.596,E2 -22951.596} C_VEL
LIN {X 0,Y 249.768,Z 384.788,A -85,B 0,C 180,E1 -22953.226,E2 -22953.226} C_VEL
LIN {X 0,Y 246.314,Z 383.873,A -85,B 0,C 180,E1 -22954.91,E2 -22954.91} C_VEL
LIN {X 0,Y 240.757,Z 382.237,A -85,B 0,C 180,E1 -22957.129,E2 -22957.129} C_VEL
LIN {X 0,Y 234.933,Z 380.208,A -85,B 0,C 180,E1 -22959.265,E2 -22959.265} C_VEL
LIN {X 0,Y 225.886,Z 376.288,A -85,B 0,C 180,E1 -22962.579,E2 -22962.579} C_VEL
LIN {X 0,Y 218.701,Z 372.232,A -85,B 0,C 180,E1 -22965.462,E2 -22965.462} C_VEL
LIN {X 0,Y 211.476,Z 366.846,A -85,B 0,C 180,E1 -22968.76,E2 -22968.76} C_VEL
LIN {X 0,Y 205.17,Z 360.504,A -85,B 0,C 180,E1 -22972.135,E2 -22972.135} C_VEL
LIN {X 0,Y 201.046,Z 354.783,A -85,B 0,C 180,E1 -22974.801,E2 -22974.801} C_VEL
LIN {X 0,Y 197.195,Z 347.316,A -85,B 0,C 180,E1 -22977.838,E2 -22977.838} C_VEL
LIN {X 0,Y 194.659,Z 340.124,A -85,B 0,C 180,E1 -22980.361,E2 -22980.361} C_VEL
LIN {X 0,Y 192.522,Z 331.63,A -85,B 0,C 180,E1 -22982.929,E2 -22982.929} C_VEL
LIN {X 0,Y 190.469,Z 324.051,A -85,B 0,C 180,E1 -22985.051,E2 -22985.051} C_VEL
LIN {X 0,Y 187.273,Z 314.97,A -85,B 0,C 180,E1 -22987.535,E2 -22987.535} C_VEL
LIN {X 0,Y 183.37,Z 306.138,A -85,B 0,C 180,E1 -22989.98,E2 -22989.98} C_VEL
LIN {X 0,Y 178.6,Z 297.001,A -85,B 0,C 180,E1 -22992.581,E2 -22992.581} C_VEL
LIN {X 0,Y 175.658,Z 292.319,A -85,B 0,C 180,E1 -22994.017,E2 -22994.017} C_VEL
LIN {X 0,Y 173.896,Z 289.144,A -85,B 0,C 180,E1 -22994.953,E2 -22994.953} C_VEL
LIN {X 0,Y 171.968,Z 286.655,A -85,B 0,C 180,E1 -22995.832,E2 -22995.832} C_VEL
LIN {X 0,Y 171.395,Z 284.636,A -85,B 0,C 180,E1 -22996.255,E2 -22996.255} C_VEL
LIN {X 0,Y 171.395,Z 284.636,A -85,B 0,C 180,E1 -23001.176,E2 -23001.176} C_VEL
LIN {X 0,Y 171.375,Z 284.638,A -85,B 0,C 180,E1 -23005.102,E2 -23005.102} C_VEL
LIN {X 0,Y 171.419,Z 284.632,A -85,B 0,C 180,E1 -23010.546,E2 -23010.546} C_VEL
LIN {X 0,Y 171.416,Z 284.626,A -85,B 0,C 180,E1 -23015.812,E2 -23015.812} C_VEL
LIN {X 0,Y 171.489,Z 284.616,A -85,B 0,C 180,E1 -23020.877,E2 -23020.877} C_VEL
LIN {X 0,Y 171.541,Z 284.61,A -85,B 0,C 180,E1 -23025.785,E2 -23025.785} C_VEL
LIN {X 0,Y 171.833,Z 284.572,A -85,B 0,C 180,E1 -23030.599,E2 -23030.599} C_VEL
LIN {X 0,Y 171.796,Z 284.573,A -85,B 0,C 180,E1 -23035.321,E2 -23035.321} C_VEL
LIN {X 0,Y 172.318,Z 284.493,A -85,B 0,C 180,E1 -23040.014,E2 -23040.014} C_VEL
LIN {X 0,Y 171.861,Z 284.578,A -85,B 0,C 180,E1 -23047.06,E2 -23047.06} C_VEL
LIN {X 0,Y 171.771,Z 284.59,A -85,B 0,C 180,E1 -23050.907,E2 -23050.907} C_VEL
LIN {X 0,Y 171.525,Z 284.621,A -85,B 0,C 180,E1 -23056.681,E2 -23056.681} C_VEL
LIN {X 0,Y 171.487,Z 284.624,A -85,B 0,C 180,E1 -23059.511,E2 -23059.511} C_VEL
LIN {X 0,Y 171.43,Z 284.632,A -85,B 0,C 180,E1 -23061.665,E2 -23061.665} C_VEL
LIN {X 0,Y 171.55,Z 285.924,A -85,B 0,C 180,E1 -23066.799,E2 -23066.799} C_VEL
LIN {X 0,Y 171.757,Z 287.177,A -85,B 0,C 180,E1 -23070.766,E2 -23070.766} C_VEL
LIN {X 0,Y 171.968,Z 288.726,A -85,B 0,C 180,E1 -23075.18,E2 -23075.18} C_VEL
LIN {X 0,Y 172.186,Z 290.211,A -85,B 0,C 180,E1 -23079.15,E2 -23079.15} C_VEL
LIN {X 0,Y 172.29,Z 292.382,A -85,B 0,C 180,E1 -23084.226,E2 -23084.226} C_VEL
LIN {X 0,Y 173.314,Z 295.426,A -85,B 0,C 180,E1 -23084.813,E2 -23084.813} C_VEL
LIN {X 0,Y 174.697,Z 297.698,A -85,B 0,C 180,E1 -23085.504,E2 -23085.504} C_VEL
LIN {X 0,Y 176.201,Z 301.402,A -85,B 0,C 180,E1 -23086.393,E2 -23086.393} C_VEL
LIN {X 0,Y 179.133,Z 309.105,A -85,B 0,C 180,E1 -23088.212,E2 -23088.212} C_VEL
LIN {X 0,Y 181.964,Z 319.626,A -85,B 0,C 180,E1 -23090.592,E2 -23090.592} C_VEL
LIN {X 0,Y 183.534,Z 328.58,A -85,B 0,C 180,E1 -23092.631,E2 -23092.631} C_VEL
LIN {X 0,Y 184.462,Z 337.633,A -85,B 0,C 180,E1 -23094.809,E2 -23094.809} C_VEL
LIN {X 0,Y 184.672,Z 346.743,A -85,B 0,C 180,E1 -23097.174,E2 -23097.174} C_VEL
LIN {X 0,Y 184.395,Z 353.364,A -85,B 0,C 180,E1 -23099.034,E2 -23099.034} C_VEL
LIN {X 0,Y 183.804,Z 357.227,A -85,B 0,C 180,E1 -23100.194,E2 -23100.194} C_VEL
LIN {X 0,Y 180.61,Z 365.779,A -85,B 0,C 180,E1 -23102.793,E2 -23102.793} C_VEL
LIN {X 0,Y 177.534,Z 373.617,A -85,B 0,C 180,E1 -23105.804,E2 -23105.804} C_VEL
LIN {X 0,Y 174.93,Z 379.767,A -85,B 0,C 180,E1 -23108.803,E2 -23108.803} C_VEL
LIN {X 0,Y 172.595,Z 385.259,A -85,B 0,C 180,E1 -23112.218,E2 -23112.218} C_VEL
LIN {X 0,Y 170.824,Z 389.587,A -85,B 0,C 180,E1 -23115.709,E2 -23115.709} C_VEL
LIN {X 0,Y 170.036,Z 391.959,A -85,B 0,C 180,E1 -23118.073,E2 -23118.073} C_VEL
LIN {X 0,Y 169.437,Z 393.763,A -85,B 0,C 180,E1 -23120.45,E2 -23120.45} C_VEL
LIN {X 0,Y 168.884,Z 396.22,A -85,B 0,C 180,E1 -23125.226,E2 -23125.226} C_VEL
LIN {X 0,Y 168.889,Z 396.815,A -85,B 0,C 180,E1 -23127.615,E2 -23127.615} C_VEL
LIN {X 0,Y 168.966,Z 396.974,A -85,B 0,C 180,E1 -23130,E2 -23130} C_VEL
LIN {X 0,Y 168.88,Z 396.755,A -85,B 0,C 180,E1 -23132.626,E2 -23132.626} C_VEL
LIN {X 0,Y 168.889,Z 396.22,A -85,B 0,C 180,E1 -23134.774,E2 -23134.774} C_VEL
LIN {X 0,Y 169.413,Z 393.762,A -85,B 0,C 180,E1 -23139.551,E2 -23139.551} C_VEL
LIN {X 0,Y 170.393,Z 390.806,A -85,B 0,C 180,E1 -23143.111,E2 -23143.111} C_VEL
LIN {X 0,Y 171.887,Z 386.813,A -85,B 0,C 180,E1 -23146.631,E2 -23146.631} C_VEL
LIN {X 0,Y 174.142,Z 381.684,A -85,B 0,C 180,E1 -23150.062,E2 -23150.062} C_VEL
LIN {X 0,Y 176.416,Z 376.423,A -85,B 0,C 180,E1 -23152.855,E2 -23152.855} C_VEL
LIN {X 0,Y 178.161,Z 372.028,A -85,B 0,C 180,E1 -23154.842,E2 -23154.842} C_VEL
LIN {X 0,Y 180.569,Z 365.777,A -85,B 0,C 180,E1 -23157.214,E2 -23157.214} C_VEL
LIN {X 0,Y 183.775,Z 357.226,A -85,B 0,C 180,E1 -23159.811,E2 -23159.811} C_VEL
LIN {X 0,Y 184.605,Z 350.13,A -85,B 0,C 180,E1 -23161.885,E2 -23161.885} C_VEL
LIN {X 0,Y 184.671,Z 346.255,A -85,B 0,C 180,E1 -23162.964,E2 -23162.964} C_VEL
LIN {X 0,Y 184.022,Z 342.079,A -85,B 0,C 180,E1 -23164.249,E2 -23164.249} C_VEL
LIN {X 0,Y 181.141,Z 335.75,A -85,B 0,C 180,E1 -23166.476,E2 -23166.476} C_VEL
LIN {X 0,Y 177.888,Z 329.217,A -85,B 0,C 180,E1 -23168.673,E2 -23168.673} C_VEL
LIN {X 0,Y 176.635,Z 324.697,A -85,B 0,C 180,E1 -23169.873,E2 -23169.873} C_VEL
LIN {X 0,Y 174.321,Z 314.463,A -85,B 0,C 180,E1 -23172.378,E2 -23172.378} C_VEL
LIN {X 0,Y 171.858,Z 306.979,A -85,B 0,C 180,E1 -23174.286,E2 -23174.286} C_VEL
LIN {X 0,Y 169.165,Z 300.742,A -85,B 0,C 180,E1 -23175.969,E2 -23175.969} C_VEL
LIN {X 0,Y 167.562,Z 297.12,A -85,B 0,C 180,E1 -23176.982,E2 -23176.982} C_VEL
LIN {X 0,Y 165.762,Z 294.239,A -85,B 0,C 180,E1 -23177.958,E2 -23177.958} C_VEL
LIN {X 0,Y 165.191,Z 292.029,A -85,B 0,C 180,E1 -23178.418,E2 -23178.418} C_VEL
LIN {X 0,Y 165.167,Z 291.28,A -85,B 0,C 180,E1 -23180.322,E2 -23180.322} C_VEL
LIN {X 0,Y 164.949,Z 289.95,A -85,B 0,C 180,E1 -23184.048,E2 -23184.048} C_VEL
LIN {X 0,Y 164.743,Z 288.237,A -85,B 0,C 180,E1 -23189.193,E2 -23189.193} C_VEL
LIN {X 0,Y 164.515,Z 286.599,A -85,B 0,C 180,E1 -23194.696,E2 -23194.696} C_VEL
LIN {X 0,Y 164.429,Z 285.507,A -85,B 0,C 180,E1 -23199.991,E2 -23199.991} C_VEL
LIN {X 0,Y 164.489,Z 285.496,A -85,B 0,C 180,E1 -23205.132,E2 -23205.132} C_VEL
LIN {X 0,Y 164.767,Z 285.461,A -85,B 0,C 180,E1 -23210.162,E2 -23210.162} C_VEL
LIN {X 0,Y 164.822,Z 285.454,A -85,B 0,C 180,E1 -23212.637,E2 -23212.637} C_VEL
LIN {X 0,Y 165.28,Z 285.368,A -85,B 0,C 180,E1 -23219.986,E2 -23219.986} C_VEL
LIN {X 0,Y 164.745,Z 285.453,A -85,B 0,C 180,E1 -23224.88,E2 -23224.88} C_VEL
LIN {X 0,Y 164.815,Z 285.455,A -85,B 0,C 180,E1 -23227.335,E2 -23227.335} C_VEL
LIN {X 0,Y 164.69,Z 285.467,A -85,B 0,C 180,E1 -23231.044,E2 -23231.044} C_VEL
LIN {X 0,Y 164.42,Z 285.504,A -85,B 0,C 180,E1 -23237.394,E2 -23237.394} C_VEL
LIN {X 0,Y 164.331,Z 285.516,A -85,B 0,C 180,E1 -23242.621,E2 -23242.621} C_VEL
LIN {X 0,Y 164.36,Z 285.507,A -85,B 0,C 180,E1 -23246.112,E2 -23246.112} C_VEL
LIN {X 0,Y 164.345,Z 285.512,A -85,B 0,C 180,E1 -23251.212,E2 -23251.212} C_VEL
LIN {X 0,Y 164.316,Z 285.518,A -85,B 0,C 180,E1 -23256.763,E2 -23256.763} C_VEL
LIN {X 0,Y 164.376,Z 285.663,A -85,B 0,C 180,E1 -23261.281,E2 -23261.281} C_VEL
LIN {X 0,Y 165.348,Z 288.362,A -85,B 0,C 180,E1 -23261.899,E2 -23261.899} C_VEL
LIN {X 0,Y 167.499,Z 290.917,A -85,B 0,C 180,E1 -23263.002,E2 -23263.002} C_VEL
LIN {X 0,Y 169.477,Z 294.253,A -85,B 0,C 180,E1 -23264.136,E2 -23264.136} C_VEL
LIN {X 0,Y 170.829,Z 296.453,A -85,B 0,C 180,E1 -23264.873,E2 -23264.873} C_VEL
LIN {X 0,Y 175.722,Z 305.12,A -85,B 0,C 180,E1 -23267.7,E2 -23267.7} C_VEL
LIN {X 0,Y 179.719,Z 313.742,A -85,B 0,C 180,E1 -23270.32,E2 -23270.32} C_VEL
LIN {X 0,Y 182.547,Z 321.296,A -85,B 0,C 180,E1 -23272.539,E2 -23272.539} C_VEL
LIN {X 0,Y 185.054,Z 329.163,A -85,B 0,C 180,E1 -23274.888,E2 -23274.888} C_VEL
LIN {X 0,Y 187.069,Z 337.939,A -85,B 0,C 180,E1 -23277.58,E2 -23277.58} C_VEL
LIN {X 0,Y 189.229,Z 346.072,A -85,B 0,C 180,E1 -23280.4,E2 -23280.4} C_VEL
LIN {X 0,Y 192.244,Z 353.498,A -85,B 0,C 180,E1 -23283.415,E2 -23283.415} C_VEL
LIN {X 0,Y 196.768,Z 360.748,A -85,B 0,C 180,E1 -23286.866,E2 -23286.866} C_VEL
LIN {X 0,Y 201.857,Z 366.493,A -85,B 0,C 180,E1 -23290.017,E2 -23290.017} C_VEL
LIN {X 0,Y 208.631,Z 371.993,A -85,B 0,C 180,E1 -23293.493,E2 -23293.493} C_VEL
LIN {X 0,Y 216.425,Z 376.599,A -85,B 0,C 180,E1 -23296.891,E2 -23296.891} C_VEL
LIN {X 0,Y 224.723,Z 380.224,A -85,B 0,C 180,E1 -23300.096,E2 -23300.096} C_VEL
LIN {X 0,Y 233.466,Z 383.053,A -85,B 0,C 180,E1 -23303.294,E2 -23303.294} C_VEL
LIN {X 0,Y 239.577,Z 384.557,A -85,B 0,C 180,E1 -23305.68,E2 -23305.68} C_VEL
LIN {X 0,Y 241.708,Z 385.011,A -85,B 0,C 180,E1 -23306.666,E2 -23306.666} C_VEL
LIN {X 0,Y 245.955,Z 385.602,A -85,B 0,C 180,E1 -23309.084,E2 -23309.084} C_VEL
LIN {X 0,Y 247.006,Z 385.624,A -85,B 0,C 180,E1 -23310,E2 -23310} C_VEL
LIN {X 0,Y 244.738,Z 385.505,A -85,B 0,C 180,E1 -23311.646,E2 -23311.646} C_VEL
LIN {X 0,Y 241.719,Z 385.01,A -85,B 0,C 180,E1 -23313.334,E2 -23313.334} C_VEL
LIN {X 0,Y 237.701,Z 384.106,A -85,B 0,C 180,E1 -23315.089,E2 -23315.089} C_VEL
LIN {X 0,Y 232.9,Z 382.881,A -85,B 0,C 180,E1 -23316.933,E2 -23316.933} C_VEL
LIN {X 0,Y 224.765,Z 380.223,A -85,B 0,C 180,E1 -23319.902,E2 -23319.902} C_VEL
LIN {X 0,Y 216.341,Z 376.553,A -85,B 0,C 180,E1 -23323.144,E2 -23323.144} C_VEL
LIN {X 0,Y 208.618,Z 371.983,A -85,B 0,C 180,E1 -23326.514,E2 -23326.514} C_VEL
LIN {X 0,Y 201.85,Z 366.507,A -85,B 0,C 180,E1 -23329.978,E2 -23329.978} C_VEL
LIN {X 0,Y 196.734,Z 360.749,A -85,B 0,C 180,E1 -23333.138,E2 -23333.138} C_VEL
LIN {X 0,Y 193.063,Z 355.019,A -85,B 0,C 180,E1 -23335.901,E2 -23335.901} C_VEL
LIN {X 0,Y 189.997,Z 348.311,A -85,B 0,C 180,E1 -23338.742,E2 -23338.742} C_VEL
LIN {X 0,Y 187.591,Z 340.342,A -85,B 0,C 180,E1 -23341.634,E2 -23341.634} C_VEL
LIN {X 0,Y 185.599,Z 331.465,A -85,B 0,C 180,E1 -23344.419,E2 -23344.419} C_VEL
LIN {X 0,Y 183.594,Z 324.49,A -85,B 0,C 180,E1 -23346.524,E2 -23346.524} C_VEL
LIN {X 0,Y 180.708,Z 316.24,A -85,B 0,C 180,E1 -23348.963,E2 -23348.963} C_VEL
LIN {X 0,Y 176.605,Z 306.915,A -85,B 0,C 180,E1 -23351.766,E2 -23351.766} C_VEL
LIN {X 0,Y 171.419,Z 297.479,A -85,B 0,C 180,E1 -23354.804,E2 -23354.804} C_VEL
LIN {X 0,Y 169.347,Z 294.074,A -85,B 0,C 180,E1 -23355.932,E2 -23355.932} C_VEL
LIN {X 0,Y 167.499,Z 290.92,A -85,B 0,C 180,E1 -23356.997,E2 -23356.997} C_VEL
LIN {X 0,Y 165.01,Z 287.715,A -85,B 0,C 180,E1 -23358.302,E2 -23358.302} C_VEL
LIN {X 0,Y 164.359,Z 285.512,A -85,B 0,C 180,E1 -23358.816,E2 -23358.816} C_VEL
LIN {X 0,Y 164.314,Z 285.516,A -85,B 0,C 180,E1 -23364.355,E2 -23364.355} C_VEL
LIN {X 0,Y 164.36,Z 285.51,A -85,B 0,C 180,E1 -23369.147,E2 -23369.147} C_VEL
LIN {X 0,Y 164.381,Z 285.501,A -85,B 0,C 180,E1 -23374.706,E2 -23374.706} C_VEL
LIN {X 0,Y 164.398,Z 285.497,A -85,B 0,C 180,E1 -23380.132,E2 -23380.132} C_VEL
LIN {X 0,Y 164.468,Z 285.489,A -85,B 0,C 180,E1 -23385.16,E2 -23385.16} C_VEL
LIN {X 0,Y 164.754,Z 285.454,A -85,B 0,C 180,E1 -23390.191,E2 -23390.191} C_VEL
LIN {X 0,Y 164.815,Z 285.455,A -85,B 0,C 180,E1 -23392.665,E2 -23392.665} C_VEL
LIN {X 0,Y 165.035,Z 285.39,A -85,B 0,C 180,E1 -23397.574,E2 -23397.574} C_VEL
LIN {X 0,Y 165.28,Z 285.368,A -85,B 0,C 180,E1 -23400.014,E2 -23400.014} C_VEL
LIN {X 0,Y 164.822,Z 285.455,A -85,B 0,C 180,E1 -23407.363,E2 -23407.363} C_VEL
LIN {X 0,Y 164.706,Z 285.47,A -85,B 0,C 180,E1 -23411.072,E2 -23411.072} C_VEL
LIN {X 0,Y 164.444,Z 285.503,A -85,B 0,C 180,E1 -23417.421,E2 -23417.421} C_VEL
LIN {X 0,Y 164.429,Z 285.504,A -85,B 0,C 180,E1 -23420.009,E2 -23420.009} C_VEL
LIN {X 0,Y 164.516,Z 286.614,A -85,B 0,C 180,E1 -23425.304,E2 -23425.304} C_VEL
LIN {X 0,Y 164.75,Z 288.44,A -85,B 0,C 180,E1 -23431.444,E2 -23431.444} C_VEL
LIN {X 0,Y 164.973,Z 290.188,A -85,B 0,C 180,E1 -23436.628,E2 -23436.628} C_VEL
LIN {X 0,Y 165.194,Z 292.066,A -85,B 0,C 180,E1 -23441.528,E2 -23441.528} C_VEL
LIN {X 0,Y 165.265,Z 292.523,A -85,B 0,C 180,E1 -23441.702,E2 -23441.702} C_VEL
LIN {X 0,Y 166.319,Z 295.393,A -85,B 0,C 180,E1 -23442.358,E2 -23442.358} C_VEL
LIN {X 0,Y 168.066,Z 298.16,A -85,B 0,C 180,E1 -23443.328,E2 -23443.328} C_VEL
LIN {X 0,Y 170.584,Z 303.888,A -85,B 0,C 180,E1 -23444.89,E2 -23444.89} C_VEL
LIN {X 0,Y 173.865,Z 312.838,A -85,B 0,C 180,E1 -23447.241,E2 -23447.241} C_VEL
LIN {X 0,Y 176.3,Z 322.826,A -85,B 0,C 180,E1 -23449.692,E2 -23449.692} C_VEL
LIN {X 0,Y 177.561,Z 331.494,A -85,B 0,C 180,E1 -23451.831,E2 -23451.831} C_VEL
LIN {X 0,Y 178.223,Z 340.173,A -85,B 0,C 180,E1 -23454.087,E2 -23454.087} C_VEL
LIN {X 0,Y 178.259,Z 347.517,A -85,B 0,C 180,E1 -23456.127,E2 -23456.127} C_VEL
LIN {X 0,Y 177.788,Z 355.094,A -85,B 0,C 180,E1 -23458.415,E2 -23458.415} C_VEL
LIN {X 0,Y 176.995,Z 358.952,A -85,B 0,C 180,E1 -23459.585,E2 -23459.585} C_VEL
LIN {X 0,Y 173.09,Z 368.532,A -85,B 0,C 180,E1 -23462.821,E2 -23462.821} C_VEL
LIN {X 0,Y 170.335,Z 375.071,A -85,B 0,C 180,E1 -23465.633,E2 -23465.633} C_VEL
LIN {X 0,Y 168.303,Z 379.571,A -85,B 0,C 180,E1 -23467.925,E2 -23467.925} C_VEL
LIN {X 0,Y 165.836,Z 385.064,A -85,B 0,C 180,E1 -23471.468,E2 -23471.468} C_VEL
LIN {X 0,Y 163.904,Z 389.391,A -85,B 0,C 180,E1 -23475.092,E2 -23475.092} C_VEL
LIN {X 0,Y 163.063,Z 391.764,A -85,B 0,C 180,E1 -23477.555,E2 -23477.555} C_VEL
LIN {X 0,Y 162.419,Z 393.568,A -85,B 0,C 180,E1 -23480.033,E2 -23480.033} C_VEL
LIN {X 0,Y 161.787,Z 396.025,A -85,B 0,C 180,E1 -23485.016,E2 -23485.016} C_VEL
LIN {X 0,Y 161.792,Z 396.694,A -85,B 0,C 180,E1 -23487.818,E2 -23487.818} C_VEL
LIN {X 0,Y 161.866,Z 396.779,A -85,B 0,C 180,E1 -23490,E2 -23490} C_VEL
LIN {X 0,Y 161.791,Z 396.621,A -85,B 0,C 180,E1 -23492.49,E2 -23492.49} C_VEL
LIN {X 0,Y 161.791,Z 396.025,A -85,B 0,C 180,E1 -23494.984,E2 -23494.984} C_VEL
LIN {X 0,Y 162.4,Z 393.567,A -85,B 0,C 180,E1 -23499.968,E2 -23499.968} C_VEL
LIN {X 0,Y 163.449,Z 390.611,A -85,B 0,C 180,E1 -23503.679,E2 -23503.679} C_VEL
LIN {X 0,Y 165.08,Z 386.617,A -85,B 0,C 180,E1 -23507.338,E2 -23507.338} C_VEL
LIN {X 0,Y 167.449,Z 381.488,A -85,B 0,C 180,E1 -23510.9,E2 -23510.9} C_VEL
LIN {X 0,Y 169.877,Z 376.228,A -85,B 0,C 180,E1 -23513.788,E2 -23513.788} C_VEL
LIN {X 0,Y 172.456,Z 369.907,A -85,B 0,C 180,E1 -23516.632,E2 -23516.632} C_VEL
LIN {X 0,Y 174.91,Z 363.955,A -85,B 0,C 180,E1 -23518.826,E2 -23518.826} C_VEL
LIN {X 0,Y 176.966,Z 358.951,A -85,B 0,C 180,E1 -23520.42,E2 -23520.42} C_VEL
LIN {X 0,Y 177.731,Z 355.092,A -85,B 0,C 180,E1 -23521.596,E2 -23521.596} C_VEL
LIN {X 0,Y 178.247,Z 348.225,A -85,B 0,C 180,E1 -23523.666,E2 -23523.666} C_VEL
LIN {X 0,Y 178.227,Z 340.173,A -85,B 0,C 180,E1 -23525.912,E2 -23525.912} C_VEL
LIN {X 0,Y 177.575,Z 331.441,A -85,B 0,C 180,E1 -23528.177,E2 -23528.177} C_VEL
LIN {X 0,Y 176.635,Z 324.697,A -85,B 0,C 180,E1 -23529.873,E2 -23529.873} C_VEL
LIN {X 0,Y 175.261,Z 320.314,A -85,B 0,C 180,E1 -23531.074,E2 -23531.074} C_VEL
LIN {X 0,Y 173.04,Z 316.595,A -85,B 0,C 180,E1 -23532.412,E2 -23532.412} C_VEL
LIN {X 0,Y 165.923,Z 307.55,A -85,B 0,C 180,E1 -23536.229,E2 -23536.229} C_VEL
LIN {X 0,Y 164.423,Z 304.897,A -85,B 0,C 180,E1 -23537.146,E2 -23537.146} C_VEL
LIN {X 0,Y 163.043,Z 301.871,A -85,B 0,C 180,E1 -23538.061,E2 -23538.061} C_VEL
LIN {X 0,Y 161.206,Z 298.202,A -85,B 0,C 180,E1 -23539.279,E2 -23539.279} C_VEL
LIN {X 0,Y 160.669,Z 297.072,A -85,B 0,C 180,E1 -23539.654,E2 -23539.654} C_VEL
LIN {X 0,Y 158.7,Z 294.166,A -85,B 0,C 180,E1 -23540.848,E2 -23540.848} C_VEL
LIN {X 0,Y 157.998,Z 291.745,A -85,B 0,C 180,E1 -23541.467,E2 -23541.467} C_VEL
LIN {X 0,Y 157.854,Z 290.688,A -85,B 0,C 180,E1 -23544.619,E2 -23544.619} C_VEL
LIN {X 0,Y 157.715,Z 289.663,A -85,B 0,C 180,E1 -23547.849,E2 -23547.849} C_VEL
LIN {X 0,Y 157.509,Z 288.03,A -85,B 0,C 180,E1 -23553.485,E2 -23553.485} C_VEL
LIN {X 0,Y 157.364,Z 286.633,A -85,B 0,C 180,E1 -23559.052,E2 -23559.052} C_VEL
LIN {X 0,Y 157.422,Z 286.377,A -85,B 0,C 180,E1 -23564.448,E2 -23564.448} C_VEL
LIN {X 0,Y 157.69,Z 286.344,A -85,B 0,C 180,E1 -23569.716,E2 -23569.716} C_VEL
LIN {X 0,Y 157.761,Z 286.334,A -85,B 0,C 180,E1 -23572.305,E2 -23572.305} C_VEL
LIN {X 0,Y 158.241,Z 286.243,A -85,B 0,C 180,E1 -23579.985,E2 -23579.985} C_VEL
LIN {X 0,Y 157.752,Z 286.333,A -85,B 0,C 180,E1 -23587.665,E2 -23587.665} C_VEL
LIN {X 0,Y 157.62,Z 286.349,A -85,B 0,C 180,E1 -23591.211,E2 -23591.211} C_VEL
LIN {X 0,Y 157.4,Z 286.371,A -85,B 0,C 180,E1 -23595.523,E2 -23595.523} C_VEL
LIN {X 0,Y 157.291,Z 286.385,A -85,B 0,C 180,E1 -23600.926,E2 -23600.926} C_VEL
LIN {X 0,Y 157.286,Z 286.391,A -85,B 0,C 180,E1 -23606.667,E2 -23606.667} C_VEL
LIN {X 0,Y 157.248,Z 286.398,A -85,B 0,C 180,E1 -23612.414,E2 -23612.414} C_VEL
LIN {X 0,Y 157.261,Z 286.396,A -85,B 0,C 180,E1 -23617.461,E2 -23617.461} C_VEL
LIN {X 0,Y 157.244,Z 286.396,A -85,B 0,C 180,E1 -23618.243,E2 -23618.243} C_VEL
LIN {X 0,Y 158.171,Z 289.11,A -85,B 0,C 180,E1 -23618.958,E2 -23618.958} C_VEL
LIN {X 0,Y 160.616,Z 291.939,A -85,B 0,C 180,E1 -23620.403,E2 -23620.403} C_VEL
LIN {X 0,Y 162.538,Z 295.204,A -85,B 0,C 180,E1 -23621.645,E2 -23621.645} C_VEL
LIN {X 0,Y 163.591,Z 296.581,A -85,B 0,C 180,E1 -23622.246,E2 -23622.246} C_VEL
LIN {X 0,Y 166.685,Z 301.955,A -85,B 0,C 180,E1 -23624.212,E2 -23624.212} C_VEL
LIN {X 0,Y 171.081,Z 310.208,A -85,B 0,C 180,E1 -23627.105,E2 -23627.105} C_VEL
LIN {X 0,Y 175.29,Z 320.247,A -85,B 0,C 180,E1 -23630.4,E2 -23630.4} C_VEL
LIN {X 0,Y 178.101,Z 329.208,A -85,B 0,C 180,E1 -23633.252,E2 -23633.252} C_VEL
LIN {X 0,Y 179.986,Z 336.75,A -85,B 0,C 180,E1 -23635.708,E2 -23635.708} C_VEL
LIN {X 0,Y 182.063,Z 346.579,A -85,B 0,C 180,E1 -23639.208,E2 -23639.208} C_VEL
LIN {X 0,Y 184.559,Z 353.75,A -85,B 0,C 180,E1 -23642.223,E2 -23642.223} C_VEL
LIN {X 0,Y 187.674,Z 359.687,A -85,B 0,C 180,E1 -23645.094,E2 -23645.094} C_VEL
LIN {X 0,Y 192.323,Z 365.933,A -85,B 0,C 180,E1 -23648.567,E2 -23648.567} C_VEL
LIN {X 0,Y 196.803,Z 370.2,A -85,B 0,C 180,E1 -23651.253,E2 -23651.253} C_VEL
LIN {X 0,Y 203.812,Z 375.144,A -85,B 0,C 180,E1 -23654.852,E2 -23654.852} C_VEL
LIN {X 0,Y 212.383,Z 379.378,A -85,B 0,C 180,E1 -23658.548,E2 -23658.548} C_VEL
LIN {X 0,Y 220.205,Z 382.172,A -85,B 0,C 180,E1 -23661.547,E2 -23661.547} C_VEL
LIN {X 0,Y 226.188,Z 383.813,A -85,B 0,C 180,E1 -23663.744,E2 -23663.744} C_VEL
LIN {X 0,Y 233.475,Z 385.239,A -85,B 0,C 180,E1 -23666.549,E2 -23666.549} C_VEL
LIN {X 0,Y 236.936,Z 385.717,A -85,B 0,C 180,E1 -23668.3,E2 -23668.3} C_VEL
LIN {X 0,Y 239.653,Z 385.822,A -85,B 0,C 180,E1 -23670,E2 -23670} C_VEL
LIN {X 0,Y 236.932,Z 385.718,A -85,B 0,C 180,E1 -23671.7,E2 -23671.7} C_VEL
LIN {X 0,Y 232.405,Z 385.057,A -85,B 0,C 180,E1 -23673.895,E2 -23673.895} C_VEL
LIN {X 0,Y 226.197,Z 383.798,A -85,B 0,C 180,E1 -23676.277,E2 -23676.277} C_VEL
LIN {X 0,Y 218.033,Z 381.497,A -85,B 0,C 180,E1 -23679.274,E2 -23679.274} C_VEL
LIN {X 0,Y 208.993,Z 377.912,A -85,B 0,C 180,E1 -23682.851,E2 -23682.851} C_VEL
LIN {X 0,Y 201.643,Z 373.812,A -85,B 0,C 180,E1 -23686.19,E2 -23686.19} C_VEL
LIN {X 0,Y 194.473,Z 368.175,A -85,B 0,C 180,E1 -23690.059,E2 -23690.059} C_VEL
LIN {X 0,Y 189.052,Z 361.83,A -85,B 0,C 180,E1 -23693.767,E2 -23693.767} C_VEL
LIN {X 0,Y 185.232,Z 355.252,A -85,B 0,C 180,E1 -23697.083,E2 -23697.083} C_VEL
LIN {X 0,Y 182.642,Z 348.535,A -85,B 0,C 180,E1 -23700.015,E2 -23700.015} C_VEL
LIN {X 0,Y 180.909,Z 341.561,A -85,B 0,C 180,E1 -23702.648,E2 -23702.648} C_VEL
LIN {X 0,Y 179.117,Z 332.942,A -85,B 0,C 180,E1 -23705.523,E2 -23705.523} C_VEL
LIN {X 0,Y 176.705,Z 324.438,A -85,B 0,C 180,E1 -23708.259,E2 -23708.259} C_VEL
LIN {X 0,Y 173.878,Z 316.786,A -85,B 0,C 180,E1 -23710.749,E2 -23710.749} C_VEL
LIN {X 0,Y 169.975,Z 308.05,A -85,B 0,C 180,E1 -23713.651,E2 -23713.651} C_VEL
LIN {X 0,Y 165.808,Z 300.103,A -85,B 0,C 180,E1 -23716.424,E2 -23716.424} C_VEL
LIN {X 0,Y 163.369,Z 296.203,A -85,B 0,C 180,E1 -23717.891,E2 -23717.891} C_VEL
LIN {X 0,Y 160.894,Z 292.633,A -85,B 0,C 180,E1 -23719.382,E2 -23719.382} C_VEL
LIN {X 0,Y 160.166,Z 291.231,A -85,B 0,C 180,E1 -23719.888,E2 -23719.888} C_VEL
LIN {X 0,Y 158.175,Z 289.092,A -85,B 0,C 180,E1 -23721.043,E2 -23721.043} C_VEL
LIN {X 0,Y 157.294,Z 286.805,A -85,B 0,C 180,E1 -23721.693,E2 -23721.693} C_VEL
LIN {X 0,Y 157.238,Z 286.397,A -85,B 0,C 180,E1 -23721.833,E2 -23721.833} C_VEL
LIN {X 0,Y 157.261,Z 286.394,A -85,B 0,C 180,E1 -23724.502,E2 -23724.502} C_VEL
LIN {X 0,Y 157.265,Z 286.395,A -85,B 0,C 180,E1 -23728.111,E2 -23728.111} C_VEL
LIN {X 0,Y 157.289,Z 286.39,A -85,B 0,C 180,E1 -23733.479,E2 -23733.479} C_VEL
LIN {X 0,Y 157.341,Z 286.376,A -85,B 0,C 180,E1 -23739.717,E2 -23739.717} C_VEL
LIN {X 0,Y 157.4,Z 286.371,A -85,B 0,C 180,E1 -23744.477,E2 -23744.477} C_VEL
LIN {X 0,Y 157.676,Z 286.336,A -85,B 0,C 180,E1 -23749.746,E2 -23749.746} C_VEL
LIN {X 0,Y 157.752,Z 286.333,A -85,B 0,C 180,E1 -23752.335,E2 -23752.335} C_VEL
LIN {X 0,Y 158.241,Z 286.243,A -85,B 0,C 180,E1 -23760.015,E2 -23760.015} C_VEL
LIN {X 0,Y 157.761,Z 286.335,A -85,B 0,C 180,E1 -23767.695,E2 -23767.695} C_VEL
LIN {X 0,Y 157.636,Z 286.351,A -85,B 0,C 180,E1 -23771.241,E2 -23771.241} C_VEL
LIN {X 0,Y 157.422,Z 286.379,A -85,B 0,C 180,E1 -23775.552,E2 -23775.552} C_VEL
LIN {X 0,Y 157.364,Z 286.631,A -85,B 0,C 180,E1 -23780.948,E2 -23780.948} C_VEL
LIN {X 0,Y 157.511,Z 288.114,A -85,B 0,C 180,E1 -23786.829,E2 -23786.829} C_VEL
LIN {X 0,Y 157.718,Z 289.722,A -85,B 0,C 180,E1 -23792.341,E2 -23792.341} C_VEL
LIN {X 0,Y 157.94,Z 291.147,A -85,B 0,C 180,E1 -23796.78,E2 -23796.78} C_VEL
LIN {X 0,Y 158.043,Z 292.073,A -85,B 0,C 180,E1 -23798.656,E2 -23798.656} C_VEL
LIN {X 0,Y 159.067,Z 294.871,A -85,B 0,C 180,E1 -23799.384,E2 -23799.384} C_VEL
LIN {X 0,Y 161.094,Z 297.786,A -85,B 0,C 180,E1 -23800.619,E2 -23800.619} C_VEL
LIN {X 0,Y 162.694,Z 301.374,A -85,B 0,C 180,E1 -23801.738,E2 -23801.738} C_VEL
LIN {X 0,Y 163.8,Z 303.392,A -85,B 0,C 180,E1 -23802.426,E2 -23802.426} C_VEL
LIN {X 0,Y 166.243,Z 309.442,A -85,B 0,C 180,E1 -23804.245,E2 -23804.245} C_VEL
LIN {X 0,Y 168.747,Z 317.07,A -85,B 0,C 180,E1 -23806.38,E2 -23806.38} C_VEL
LIN {X 0,Y 170.819,Z 327.225,A -85,B 0,C 180,E1 -23809.084,E2 -23809.084} C_VEL
LIN {X 0,Y 171.758,Z 337.24,A -85,B 0,C 180,E1 -23811.773,E2 -23811.773} C_VEL
LIN {X 0,Y 172.017,Z 346.277,A -85,B 0,C 180,E1 -23814.397,E2 -23814.397} C_VEL
LIN {X 0,Y 171.467,Z 354.902,A -85,B 0,C 180,E1 -23817.112,E2 -23817.112} C_VEL
LIN {X 0,Y 170.829,Z 358.755,A -85,B 0,C 180,E1 -23818.363,E2 -23818.363} C_VEL
LIN {X 0,Y 166.772,Z 368.336,A -85,B 0,C 180,E1 -23821.701,E2 -23821.701} C_VEL
LIN {X 0,Y 163.849,Z 374.875,A -85,B 0,C 180,E1 -23824.601,E2 -23824.601} C_VEL
LIN {X 0,Y 161.73,Z 379.376,A -85,B 0,C 180,E1 -23826.978,E2 -23826.978} C_VEL
LIN {X 0,Y 159.083,Z 384.869,A -85,B 0,C 180,E1 -23830.651,E2 -23830.651} C_VEL
LIN {X 0,Y 157.009,Z 389.195,A -85,B 0,C 180,E1 -23834.421,E2 -23834.421} C_VEL
LIN {X 0,Y 156.089,Z 391.568,A -85,B 0,C 180,E1 -23836.99,E2 -23836.99} C_VEL
LIN {X 0,Y 155.421,Z 393.373,A -85,B 0,C 180,E1 -23839.579,E2 -23839.579} C_VEL
LIN {X 0,Y 154.717,Z 395.83,A -85,B 0,C 180,E1 -23844.788,E2 -23844.788} C_VEL
LIN {X 0,Y 154.696,Z 396.581,A -85,B 0,C 180,E1 -23848.571,E2 -23848.571} C_VEL
LIN {X 0,Y 154.696,Z 396.426,A -85,B 0,C 180,E1 -23852.604,E2 -23852.604} C_VEL
LIN {X 0,Y 154.719,Z 395.83,A -85,B 0,C 180,E1 -23855.212,E2 -23855.212} C_VEL
LIN {X 0,Y 155.377,Z 393.371,A -85,B 0,C 180,E1 -23860.424,E2 -23860.424} C_VEL
LIN {X 0,Y 156.527,Z 390.415,A -85,B 0,C 180,E1 -23864.297,E2 -23864.297} C_VEL
LIN {X 0,Y 158.306,Z 386.422,A -85,B 0,C 180,E1 -23868.105,E2 -23868.105} C_VEL
LIN {X 0,Y 160.785,Z 381.292,A -85,B 0,C 180,E1 -23871.81,E2 -23871.81} C_VEL
LIN {X 0,Y 163.36,Z 376.032,A -85,B 0,C 180,E1 -23874.8,E2 -23874.8} C_VEL
LIN {X 0,Y 165.408,Z 371.329,A -85,B 0,C 180,E1 -23877.057,E2 -23877.057} C_VEL
LIN {X 0,Y 168.007,Z 365.386,A -85,B 0,C 180,E1 -23879.44,E2 -23879.44} C_VEL
LIN {X 0,Y 170.787,Z 358.754,A -85,B 0,C 180,E1 -23881.645,E2 -23881.645} C_VEL
LIN {X 0,Y 171.809,Z 350.922,A -85,B 0,C 180,E1 -23884.205,E2 -23884.205} C_VEL
LIN {X 0,Y 172.008,Z 341.328,A -85,B 0,C 180,E1 -23887.059,E2 -23887.059} C_VEL
LIN {X 0,Y 171.339,Z 331.757,A -85,B 0,C 180,E1 -23889.712,E2 -23889.712} C_VEL
LIN {X 0,Y 170.122,Z 323.382,A -85,B 0,C 180,E1 -23891.944,E2 -23891.944} C_VEL
LIN {X 0,Y 167.733,Z 313.629,A -85,B 0,C 180,E1 -23894.561,E2 -23894.561} C_VEL
LIN {X 0,Y 164.63,Z 305.349,A -85,B 0,C 180,E1 -23897.007,E2 -23897.007} C_VEL
LIN {X 0,Y 164.423,Z 304.897,A -85,B 0,C 180,E1 -23897.146,E2 -23897.146} C_VEL
LIN {X 0,Y 162.766,Z 302.56,A -85,B 0,C 180,E1 -23898.093,E2 -23898.093} C_VEL
LIN {X 0,Y 159.192,Z 300.07,A -85,B 0,C 180,E1 -23899.873,E2 -23899.873} C_VEL
LIN {X 0,Y 154.673,Z 297.712,A -85,B 0,C 180,E1 -23902.21,E2 -23902.21} C_VEL
LIN {X 0,Y 153.347,Z 296.667,A -85,B 0,C 180,E1 -23903.004,E2 -23903.004} C_VEL
LIN {X 0,Y 151.479,Z 293.859,A -85,B 0,C 180,E1 -23904.332,E2 -23904.332} C_VEL
LIN {X 0,Y 150.775,Z 291.499,A -85,B 0,C 180,E1 -23904.96,E2 -23904.96} C_VEL
LIN {X 0,Y 150.588,Z 290.284,A -85,B 0,C 180,E1 -23909.095,E2 -23909.095} C_VEL
LIN {X 0,Y 150.5,Z 289.34,A -85,B 0,C 180,E1 -23912.528,E2 -23912.528} C_VEL
LIN {X 0,Y 150.342,Z 287.993,A -85,B 0,C 180,E1 -23918.024,E2 -23918.024} C_VEL
LIN {X 0,Y 150.33,Z 287.367,A -85,B 0,C 180,E1 -23920.882,E2 -23920.882} C_VEL
LIN {X 0,Y 150.419,Z 287.249,A -85,B 0,C 180,E1 -23926.475,E2 -23926.475} C_VEL
LIN {X 0,Y 150.611,Z 287.225,A -85,B 0,C 180,E1 -23929.227,E2 -23929.227} C_VEL
LIN {X 0,Y 150.7,Z 287.214,A -85,B 0,C 180,E1 -23931.942,E2 -23931.942} C_VEL
LIN {X 0,Y 151.201,Z 287.118,A -85,B 0,C 180,E1 -23939.984,E2 -23939.984} C_VEL
LIN {X 0,Y 150.69,Z 287.211,A -85,B 0,C 180,E1 -23948.027,E2 -23948.027} C_VEL
LIN {X 0,Y 150.562,Z 287.229,A -85,B 0,C 180,E1 -23951.414,E2 -23951.414} C_VEL
LIN {X 0,Y 150.304,Z 287.26,A -85,B 0,C 180,E1 -23956.276,E2 -23956.276} C_VEL
LIN {X 0,Y 150.265,Z 287.259,A -85,B 0,C 180,E1 -23960.709,E2 -23960.709} C_VEL
LIN {X 0,Y 150.217,Z 287.274,A -85,B 0,C 180,E1 -23967.264,E2 -23967.264} C_VEL
LIN {X 0,Y 150.188,Z 287.276,A -85,B 0,C 180,E1 -23972.618,E2 -23972.618} C_VEL
LIN {X 0,Y 150.186,Z 287.278,A -85,B 0,C 180,E1 -23974.751,E2 -23974.751} C_VEL
LIN {X 0,Y 151.06,Z 289.815,A -85,B 0,C 180,E1 -23975.538,E2 -23975.538} C_VEL
LIN {X 0,Y 153.143,Z 292.171,A -85,B 0,C 180,E1 -23976.983,E2 -23976.983} C_VEL
LIN {X 0,Y 153.717,Z 292.939,A -85,B 0,C 180,E1 -23977.39,E2 -23977.39} C_VEL
LIN {X 0,Y 155.438,Z 295.926,A -85,B 0,C 180,E1 -23978.672,E2 -23978.672} C_VEL
LIN {X 0,Y 156.926,Z 297.84,A -85,B 0,C 180,E1 -23979.635,E2 -23979.635} C_VEL
LIN {X 0,Y 161.753,Z 305.967,A -85,B 0,C 180,E1 -23983.074,E2 -23983.074} C_VEL
LIN {X 0,Y 165.703,Z 313.987,A -85,B 0,C 180,E1 -23986.115,E2 -23986.115} C_VEL
LIN {X 0,Y 169.03,Z 322.245,A -85,B 0,C 180,E1 -23989.057,E2 -23989.057} C_VEL
LIN {X 0,Y 171.443,Z 329.916,A -85,B 0,C 180,E1 -23991.707,E2 -23991.707} C_VEL
LIN {X 0,Y 173.498,Z 338.119,A -85,B 0,C 180,E1 -23994.605,E2 -23994.605} C_VEL
LIN {X 0,Y 175.089,Z 347.032,A -85,B 0,C 180,E1 -23997.923,E2 -23997.923} C_VEL
LIN {X 0,Y 176.995,Z 353.773,A -85,B 0,C 180,E1 -24000.842,E2 -24000.842} C_VEL
LIN {X 0,Y 179.762,Z 360.136,A -85,B 0,C 180,E1 -24004.017,E2 -24004.017} C_VEL
LIN {X 0,Y 183.852,Z 366.178,A -85,B 0,C 180,E1 -24007.527,E2 -24007.527} C_VEL
LIN {X 0,Y 189.296,Z 371.639,A -85,B 0,C 180,E1 -24011.212,E2 -24011.212} C_VEL
LIN {X 0,Y 196.36,Z 376.46,A -85,B 0,C 180,E1 -24015.039,E2 -24015.039} C_VEL
LIN {X 0,Y 202.828,Z 379.641,A -85,B 0,C 180,E1 -24018.001,E2 -24018.001} C_VEL
LIN {X 0,Y 208.433,Z 381.764,A -85,B 0,C 180,E1 -24020.294,E2 -24020.294} C_VEL
LIN {X 0,Y 214.088,Z 383.4,A -85,B 0,C 180,E1 -24022.455,E2 -24022.455} C_VEL
LIN {X 0,Y 219.615,Z 384.597,A -85,B 0,C 180,E1 -24024.491,E2 -24024.491} C_VEL
LIN {X 0,Y 225.235,Z 385.541,A -85,B 0,C 180,E1 -24026.611,E2 -24026.611} C_VEL
LIN {X 0,Y 228.895,Z 385.937,A -85,B 0,C 180,E1 -24028.241,E2 -24028.241} C_VEL
LIN {X 0,Y 232.152,Z 386.024,A -85,B 0,C 180,E1 -24030,E2 -24030} C_VEL
LIN {X 0,Y 228.9,Z 385.937,A -85,B 0,C 180,E1 -24031.759,E2 -24031.759} C_VEL
LIN {X 0,Y 224.783,Z 385.478,A -85,B 0,C 180,E1 -24033.585,E2 -24033.585} C_VEL
LIN {X 0,Y 218.93,Z 384.451,A -85,B 0,C 180,E1 -24035.788,E2 -24035.788} C_VEL
LIN {X 0,Y 212.868,Z 383.038,A -85,B 0,C 180,E1 -24038.02,E2 -24038.02} C_VEL
LIN {X 0,Y 207.069,Z 381.287,A -85,B 0,C 180,E1 -24040.259,E2 -24040.259} C_VEL
LIN {X 0,Y 197.44,Z 377.078,A -85,B 0,C 180,E1 -24044.428,E2 -24044.428} C_VEL
LIN {X 0,Y 191.528,Z 373.396,A -85,B 0,C 180,E1 -24047.488,E2 -24047.488} C_VEL
LIN {X 0,Y 185.753,Z 368.361,A -85,B 0,C 180,E1 -24051.077,E2 -24051.077} C_VEL
LIN {X 0,Y 181.187,Z 362.554,A -85,B 0,C 180,E1 -24054.643,E2 -24054.643} C_VEL
LIN {X 0,Y 178.258,Z 357.06,A -85,B 0,C 180,E1 -24057.596,E2 -24057.596} C_VEL
LIN {X 0,Y 175.982,Z 350.57,A -85,B 0,C 180,E1 -24060.628,E2 -24060.628} C_VEL
LIN {X 0,Y 174.122,Z 341.781,A -85,B 0,C 180,E1 -24064.089,E2 -24064.089} C_VEL
LIN {X 0,Y 172.51,Z 333.743,A -85,B 0,C 180,E1 -24066.945,E2 -24066.945} C_VEL
LIN {X 0,Y 169.915,Z 324.845,A -85,B 0,C 180,E1 -24070.048,E2 -24070.048} C_VEL
LIN {X 0,Y 166.451,Z 315.685,A -85,B 0,C 180,E1 -24073.276,E2 -24073.276} C_VEL
LIN {X 0,Y 161.741,Z 306.017,A -85,B 0,C 180,E1 -24076.922,E2 -24076.922} C_VEL
LIN {X 0,Y 156.73,Z 297.423,A -85,B 0,C 180,E1 -24080.514,E2 -24080.514} C_VEL
LIN {X 0,Y 154.216,Z 294.078,A -85,B 0,C 180,E1 -24082.19,E2 -24082.19} C_VEL
LIN {X 0,Y 153.285,Z 292.271,A -85,B 0,C 180,E1 -24082.931,E2 -24082.931} C_VEL
LIN {X 0,Y 151.161,Z 289.974,A -85,B 0,C 180,E1 -24084.387,E2 -24084.387} C_VEL
LIN {X 0,Y 150.248,Z 287.726,A -85,B 0,C 180,E1 -24085.164,E2 -24085.164} C_VEL
LIN {X 0,Y 150.191,Z 287.278,A -85,B 0,C 180,E1 -24085.352,E2 -24085.352} C_VEL
LIN {X 0,Y 150.178,Z 287.276,A -85,B 0,C 180,E1 -24089.038,E2 -24089.038} C_VEL
LIN {X 0,Y 150.217,Z 287.274,A -85,B 0,C 180,E1 -24092.736,E2 -24092.736} C_VEL
LIN {X 0,Y 150.265,Z 287.259,A -85,B 0,C 180,E1 -24099.291,E2 -24099.291} C_VEL
LIN {X 0,Y 150.304,Z 287.26,A -85,B 0,C 180,E1 -24103.724,E2 -24103.724} C_VEL
LIN {X 0,Y 150.595,Z 287.22,A -85,B 0,C 180,E1 -24109.258,E2 -24109.258} C_VEL
LIN {X 0,Y 150.69,Z 287.211,A -85,B 0,C 180,E1 -24111.973,E2 -24111.973} C_VEL
LIN {X 0,Y 151.201,Z 287.118,A -85,B 0,C 180,E1 -24120.016,E2 -24120.016} C_VEL
LIN {X 0,Y 150.7,Z 287.215,A -85,B 0,C 180,E1 -24128.058,E2 -24128.058} C_VEL
LIN {X 0,Y 150.578,Z 287.231,A -85,B 0,C 180,E1 -24131.444,E2 -24131.444} C_VEL
LIN {X 0,Y 150.327,Z 287.262,A -85,B 0,C 180,E1 -24136.306,E2 -24136.306} C_VEL
LIN {X 0,Y 150.33,Z 287.365,A -85,B 0,C 180,E1 -24139.118,E2 -24139.118} C_VEL
LIN {X 0,Y 150.419,Z 288.679,A -85,B 0,C 180,E1 -24144.882,E2 -24144.882} C_VEL
LIN {X 0,Y 150.504,Z 289.442,A -85,B 0,C 180,E1 -24147.853,E2 -24147.853} C_VEL
LIN {X 0,Y 150.684,Z 290.863,A -85,B 0,C 180,E1 -24152.911,E2 -24152.911} C_VEL
LIN {X 0,Y 150.802,Z 291.586,A -85,B 0,C 180,E1 -24155.033,E2 -24155.033} C_VEL
LIN {X 0,Y 151.879,Z 294.663,A -85,B 0,C 180,E1 -24155.968,E2 -24155.968} C_VEL
LIN {X 0,Y 154.256,Z 297.904,A -85,B 0,C 180,E1 -24157.624,E2 -24157.624} C_VEL
LIN {X 0,Y 155.926,Z 301.393,A -85,B 0,C 180,E1 -24158.913,E2 -24158.913} C_VEL
LIN {X 0,Y 157.098,Z 303.451,A -85,B 0,C 180,E1 -24159.727,E2 -24159.727} C_VEL
LIN {X 0,Y 160.031,Z 310.024,A -85,B 0,C 180,E1 -24162.062,E2 -24162.062} C_VEL
LIN {X 0,Y 162.577,Z 317.391,A -85,B 0,C 180,E1 -24164.392,E2 -24164.392} C_VEL
LIN {X 0,Y 164.724,Z 327.734,A -85,B 0,C 180,E1 -24167.405,E2 -24167.405} C_VEL
LIN {X 0,Y 165.576,Z 336.231,A -85,B 0,C 180,E1 -24169.838,E2 -24169.838} C_VEL
LIN {X 0,Y 165.797,Z 344.964,A -85,B 0,C 180,E1 -24172.476,E2 -24172.476} C_VEL
LIN {X 0,Y 165.309,Z 353.3,A -85,B 0,C 180,E1 -24175.189,E2 -24175.189} C_VEL
LIN {X 0,Y 164.627,Z 358.554,A -85,B 0,C 180,E1 -24177.024,E2 -24177.024} C_VEL
LIN {X 0,Y 162.589,Z 363.565,A -85,B 0,C 180,E1 -24178.755,E2 -24178.755} C_VEL
LIN {X 0,Y 159.867,Z 369.517,A -85,B 0,C 180,E1 -24181.082,E2 -24181.082} C_VEL
LIN {X 0,Y 157.409,Z 374.678,A -85,B 0,C 180,E1 -24183.483,E2 -24183.483} C_VEL
LIN {X 0,Y 155.211,Z 379.181,A -85,B 0,C 180,E1 -24185.951,E2 -24185.951} C_VEL
LIN {X 0,Y 152.374,Z 384.673,A -85,B 0,C 180,E1 -24189.762,E2 -24189.762} C_VEL
LIN {X 0,Y 150.143,Z 388.999,A -85,B 0,C 180,E1 -24193.689,E2 -24193.689} C_VEL
LIN {X 0,Y 149.144,Z 391.372,A -85,B 0,C 180,E1 -24196.373,E2 -24196.373} C_VEL
LIN {X 0,Y 148.408,Z 393.177,A -85,B 0,C 180,E1 -24199.081,E2 -24199.081} C_VEL
LIN {X 0,Y 147.646,Z 395.636,A -85,B 0,C 180,E1 -24204.537,E2 -24204.537} C_VEL
LIN {X 0,Y 147.638,Z 396.388,A -85,B 0,C 180,E1 -24209.11,E2 -24209.11} C_VEL
LIN {X 0,Y 147.599,Z 396.231,A -85,B 0,C 180,E1 -24212.729,E2 -24212.729} C_VEL
LIN {X 0,Y 147.647,Z 395.636,A -85,B 0,C 180,E1 -24215.463,E2 -24215.463} C_VEL
LIN {X 0,Y 148.373,Z 393.176,A -85,B 0,C 180,E1 -24220.922,E2 -24220.922} C_VEL
LIN {X 0,Y 149.63,Z 390.22,A -85,B 0,C 180,E1 -24224.971,E2 -24224.971} C_VEL
LIN {X 0,Y 151.561,Z 386.227,A -85,B 0,C 180,E1 -24228.941,E2 -24228.941} C_VEL
LIN {X 0,Y 154.173,Z 381.096,A -85,B 0,C 180,E1 -24232.797,E2 -24232.797} C_VEL
LIN {X 0,Y 156.908,Z 375.836,A -85,B 0,C 180,E1 -24235.893,E2 -24235.893} C_VEL
LIN {X 0,Y 159.799,Z 369.514,A -85,B 0,C 180,E1 -24238.932,E2 -24238.932} C_VEL
LIN {X 0,Y 162.57,Z 363.565,A -85,B 0,C 180,E1 -24241.249,E2 -24241.249} C_VEL
LIN {X 0,Y 164.051,Z 360.311,A -85,B 0,C 180,E1 -24242.377,E2 -24242.377} C_VEL
LIN {X 0,Y 165.121,Z 354.977,A -85,B 0,C 180,E1 -24244.216,E2 -24244.216} C_VEL
LIN {X 0,Y 165.691,Z 347.222,A -85,B 0,C 180,E1 -24246.802,E2 -24246.802} C_VEL
LIN {X 0,Y 165.722,Z 340.011,A -85,B 0,C 180,E1 -24249.032,E2 -24249.032} C_VEL
LIN {X 0,Y 165.263,Z 332.351,A -85,B 0,C 180,E1 -24251.284,E2 -24251.284} C_VEL
LIN {X 0,Y 163.997,Z 323.643,A -85,B 0,C 180,E1 -24253.794,E2 -24253.794} C_VEL
LIN {X 0,Y 161.814,Z 314.933,A -85,B 0,C 180,E1 -24256.393,E2 -24256.393} C_VEL
LIN {X 0,Y 158.653,Z 306.68,A -85,B 0,C 180,E1 -24259.101,E2 -24259.101} C_VEL
LIN {X 0,Y 156.388,Z 302.025,A -85,B 0,C 180,E1 -24260.788,E2 -24260.788} C_VEL
LIN {X 0,Y 154.413,Z 298.351,A -85,B 0,C 180,E1 -24262.234,E2 -24262.234} C_VEL
LIN {X 0,Y 153.909,Z 297.212,A -85,B 0,C 180,E1 -24262.647,E2 -24262.647} C_VEL
LIN {X 0,Y 153.347,Z 296.667,A -85,B 0,C 180,E1 -24263.004,E2 -24263.004} C_VEL
LIN {X 0,Y 149.456,Z 293.725,A -85,B 0,C 180,E1 -24265.489,E2 -24265.489} C_VEL
LIN {X 0,Y 143.986,Z 291.32,A -85,B 0,C 180,E1 -24269.101,E2 -24269.101} C_VEL
LIN {X 0,Y 143.494,Z 291.034,A -85,B 0,C 180,E1 -24269.969,E2 -24269.969} C_VEL
LIN {X 0,Y 143.399,Z 290.063,A -85,B 0,C 180,E1 -24273.81,E2 -24273.81} C_VEL
LIN {X 0,Y 143.335,Z 288.696,A -85,B 0,C 180,E1 -24279.91,E2 -24279.91} C_VEL
LIN {X 0,Y 143.247,Z 288.143,A -85,B 0,C 180,E1 -24282.864,E2 -24282.864} C_VEL
LIN {X 0,Y 143.538,Z 288.106,A -85,B 0,C 180,E1 -24288.69,E2 -24288.69} C_VEL
LIN {X 0,Y 143.622,Z 288.096,A -85,B 0,C 180,E1 -24291.542,E2 -24291.542} C_VEL
LIN {X 0,Y 144.158,Z 287.993,A -85,B 0,C 180,E1 -24299.984,E2 -24299.984} C_VEL
LIN {X 0,Y 143.611,Z 288.09,A -85,B 0,C 180,E1 -24308.425,E2 -24308.425} C_VEL
LIN {X 0,Y 143.488,Z 288.111,A -85,B 0,C 180,E1 -24311.601,E2 -24311.601} C_VEL
LIN {X 0,Y 143.242,Z 288.143,A -85,B 0,C 180,E1 -24317.102,E2 -24317.102} C_VEL
LIN {X 0,Y 143.206,Z 288.141,A -85,B 0,C 180,E1 -24321.184,E2 -24321.184} C_VEL
LIN {X 0,Y 143.164,Z 288.151,A -85,B 0,C 180,E1 -24327.919,E2 -24327.919} C_VEL
LIN {X 0,Y 143.124,Z 288.156,A -85,B 0,C 180,E1 -24330.504,E2 -24330.504} C_VEL
LIN {X 0,Y 144.029,Z 290.8,A -85,B 0,C 180,E1 -24331.514,E2 -24331.514} C_VEL
LIN {X 0,Y 146.19,Z 293.157,A -85,B 0,C 180,E1 -24333.314,E2 -24333.314} C_VEL
LIN {X 0,Y 146.864,Z 293.855,A -85,B 0,C 180,E1 -24333.842,E2 -24333.842} C_VEL
LIN {X 0,Y 148.616,Z 296.956,A -85,B 0,C 180,E1 -24335.379,E2 -24335.379} C_VEL
LIN {X 0,Y 150.159,Z 298.788,A -85,B 0,C 180,E1 -24336.511,E2 -24336.511} C_VEL
LIN {X 0,Y 151.724,Z 301.533,A -85,B 0,C 180,E1 -24337.832,E2 -24337.832} C_VEL
LIN {X 0,Y 154.79,Z 306.516,A -85,B 0,C 180,E1 -24340.293,E2 -24340.293} C_VEL
LIN {X 0,Y 158.462,Z 313.684,A -85,B 0,C 180,E1 -24343.404,E2 -24343.404} C_VEL
LIN {X 0,Y 161.807,Z 321.391,A -85,B 0,C 180,E1 -24346.501,E2 -24346.501} C_VEL
LIN {X 0,Y 164.64,Z 329.771,A -85,B 0,C 180,E1 -24349.697,E2 -24349.697} C_VEL
LIN {X 0,Y 166.862,Z 338.805,A -85,B 0,C 180,E1 -24353.126,E2 -24353.126} C_VEL
LIN {X 0,Y 168.114,Z 346.428,A -85,B 0,C 180,E1 -24356.105,E2 -24356.105} C_VEL
LIN {X 0,Y 169.729,Z 354.132,A -85,B 0,C 180,E1 -24359.522,E2 -24359.522} C_VEL
LIN {X 0,Y 171.908,Z 360.135,A -85,B 0,C 180,E1 -24362.618,E2 -24362.618} C_VEL
LIN {X 0,Y 175.538,Z 366.42,A -85,B 0,C 180,E1 -24366.399,E2 -24366.399} C_VEL
LIN {X 0,Y 179.747,Z 371.224,A -85,B 0,C 180,E1 -24369.734,E2 -24369.734} C_VEL
LIN {X 0,Y 186.097,Z 376.119,A -85,B 0,C 180,E1 -24373.726,E2 -24373.726} C_VEL
LIN {X 0,Y 194.11,Z 380.232,A -85,B 0,C 180,E1 -24377.768,E2 -24377.768} C_VEL
LIN {X 0,Y 199.664,Z 382.289,A -85,B 0,C 180,E1 -24380.166,E2 -24380.166} C_VEL
LIN {X 0,Y 205.526,Z 383.908,A -85,B 0,C 180,E1 -24382.48,E2 -24382.48} C_VEL
LIN {X 0,Y 211.668,Z 385.105,A -85,B 0,C 180,E1 -24384.767,E2 -24384.767} C_VEL
LIN {X 0,Y 218.082,Z 385.938,A -85,B 0,C 180,E1 -24387.158,E2 -24387.158} C_VEL
LIN {X 0,Y 220.535,Z 386.165,A -85,B 0,C 180,E1 -24388.174,E2 -24388.174} C_VEL
LIN {X 0,Y 224.308,Z 386.235,A -85,B 0,C 180,E1 -24390,E2 -24390} C_VEL
LIN {X 0,Y 220.568,Z 386.164,A -85,B 0,C 180,E1 -24391.826,E2 -24391.826} C_VEL
LIN {X 0,Y 215.745,Z 385.727,A -85,B 0,C 180,E1 -24393.735,E2 -24393.735} C_VEL
LIN {X 0,Y 210.298,Z 384.85,A -85,B 0,C 180,E1 -24395.754,E2 -24395.754} C_VEL
LIN {X 0,Y 204.565,Z 383.66,A -85,B 0,C 180,E1 -24397.899,E2 -24397.899} C_VEL
